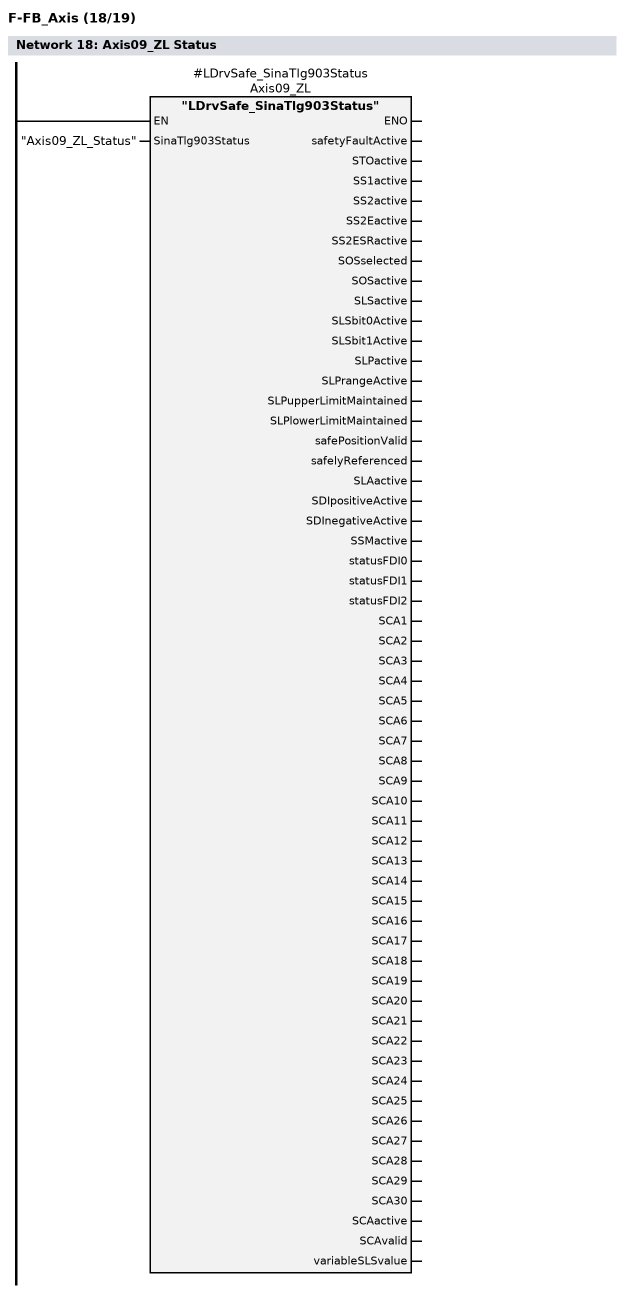
   RUNG wire#powerrail
      #LDrvSafe_SinaTlg903StatusAxis09_ZL(SinaTlg903Status := "Axis09_ZL_Status", safetyFaultActive =>, STOactive =>, SS1active =>, SS2active =>, SS2Eactive =>, SS2ESRactive =>, SOSselected =>, SOSactive =>, SLSactive =>, SLSbit0Active =>, SLSbit1Active =>, SLPactive =>, SLPrangeActive =>, SLPupperLimitMaintained =>, SLPlowerLimitMaintained =>, safePositionValid =>, safelyReferenced =>, SLAactive =>, SDIpositiveActive =>, SDInegativeActive =>, SSMactive =>, statusFDI0 =>, statusFDI1 =>, statusFDI2 =>, SCA1 =>, SCA2 =>, SCA3 =>, SCA4 =>, SCA5 =>, SCA6 =>, SCA7 =>, SCA8 =>, SCA9 =>, SCA10 =>, SCA11 =>, SCA12 =>, SCA13 =>, SCA14 =>, SCA15 =>, SCA16 =>, SCA17 =>, SCA18 =>, SCA19 =>, SCA20 =>, SCA21 =>, SCA22 =>, SCA23 =>, SCA24 =>, SCA25 =>, SCA26 =>, SCA27 =>, SCA28 =>, SCA29 =>, SCA30 =>, SCAactive =>, SCAvalid =>, variableSLSvalue =>)
   END_RUNG
   // the same network as SCL:
   #LDrvSafe_SinaTlg903StatusAxis09_ZL(SinaTlg903Status := "Axis09_ZL_Status");   // "LDrvSafe_SinaTlg903Status"
END_REGION

REGION Network 19: Axis09_ZL Control
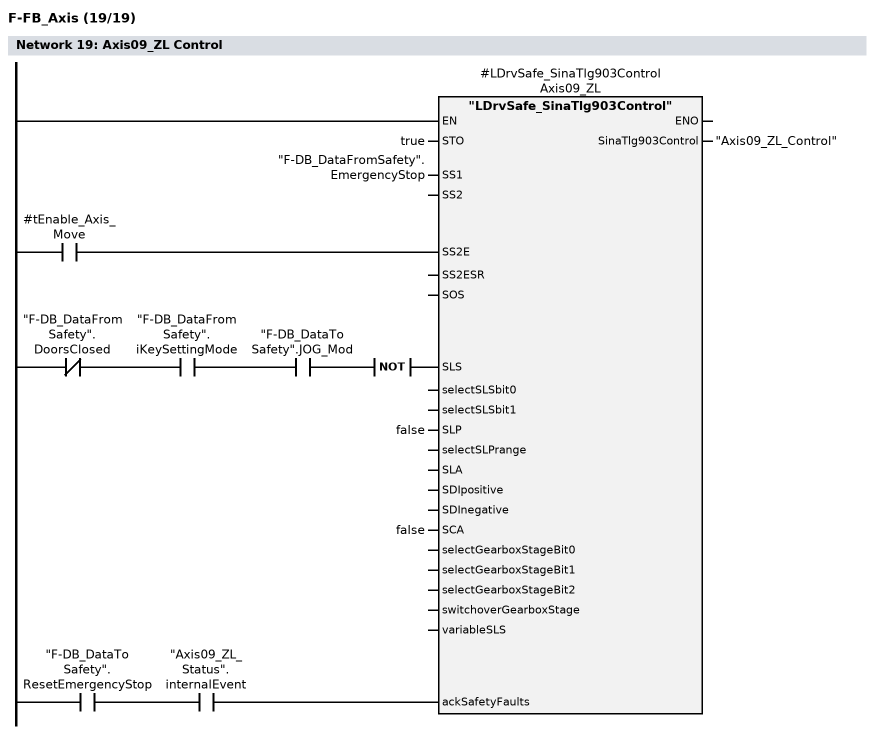
   RUNG wire#powerrail
      #LDrvSafe_SinaTlg903ControlAxis09_ZL(SS2E := wire#w1, SLS := wire#w2, ackSafetyFaults := wire#w3, STO := true, SS1 := "F-DB_DataFromSafety".EmergencyStop, SS2 :=, SS2ESR :=, SOS :=, selectSLSbit0 :=, selectSLSbit1 :=, SLP := false, selectSLPrange :=, SLA :=, SDIpositive :=, SDInegative :=, SCA := false, selectGearboxStageBit0 :=, selectGearboxStageBit1 :=, selectGearboxStageBit2 :=, switchoverGearboxStage :=, variableSLS :=, SinaTlg903Control => "Axis09_ZL_Control")
   END_RUNG
   RUNG wire#powerrail
      Contact( #tEnable_Axis_Move )
   END_RUNG wire#w1
   RUNG wire#powerrail
      I_Contact( "F-DB_DataFromSafety".DoorsClosed )
      Contact( "F-DB_DataFromSafety".iKeySettingMode )
      Contact( "F-DB_DataToSafety".JOG_Mod )
      Not()
   END_RUNG wire#w2
   RUNG wire#powerrail
      Contact( "F-DB_DataToSafety".ResetEmergencyStop )
      Contact( "Axis09_ZL_Status".internalEvent )
   END_RUNG wire#w3
   // the same network as SCL:
   #LDrvSafe_SinaTlg903ControlAxis09_ZL(STO := true,   // "LDrvSafe_SinaTlg903Control"
                           SS1 := "F-DB_DataFromSafety".EmergencyStop,
                           SS2E := #tEnable_Axis_Move,
                           SLS := NOT (NOT "F-DB_DataFromSafety".DoorsClosed AND "F-DB_DataFromSafety".iKeySettingMode AND "F-DB_DataToSafety".JOG_Mod),
                           SLP := false,
                           SCA := false,
                           ackSafetyFaults := "F-DB_DataToSafety".ResetEmergencyStop AND "Axis09_ZL_Status".internalEvent,
                           SinaTlg903Control => "Axis09_ZL_Control");
END_REGION
END_FUNCTION_BLOCK

FUNCTION_BLOCK "F-FB_Laser"   // FB140, F_LAD
{ S7_Optimized_Access := 'TRUE' }
// stored: AutoNumber false
   VAR
      FDBACK_LaserPowerSupply : FDBACK;
      FDBACK_Shutter : FDBACK;
      sFeedBackShutter : Bool;
      sAckFdbShutter : Bool;
      sLaserSupplyPower : Bool;
      sAckFdbPowLaser : Bool;
      sPositiveFrontButtonShutter : Bool;
      sNegativeFrontMaintenanceDoor : Bool;
      sNegativeFrontDoor : Bool;
      sNegativeRoofLeftDoor : Bool;
      sNegativeRoofRightDoor : Bool;
      sNegativeLaserExternDoor : Bool;
      sNegativeSasOneDoor : Bool;
   END_VAR
   VAR_TEMP   // added for the SCL form of the ladder/FBD networks
      _w1 : Bool;
      _w2 : Bool;
      _w3 : Bool;
      _w4 : Bool;
      _w5 : Bool;
      _w6 : Bool;
      _w7 : Bool;
   END_VAR
BEGIN

REGION Network 1: Laser shutter setting mode, allow opening shutter
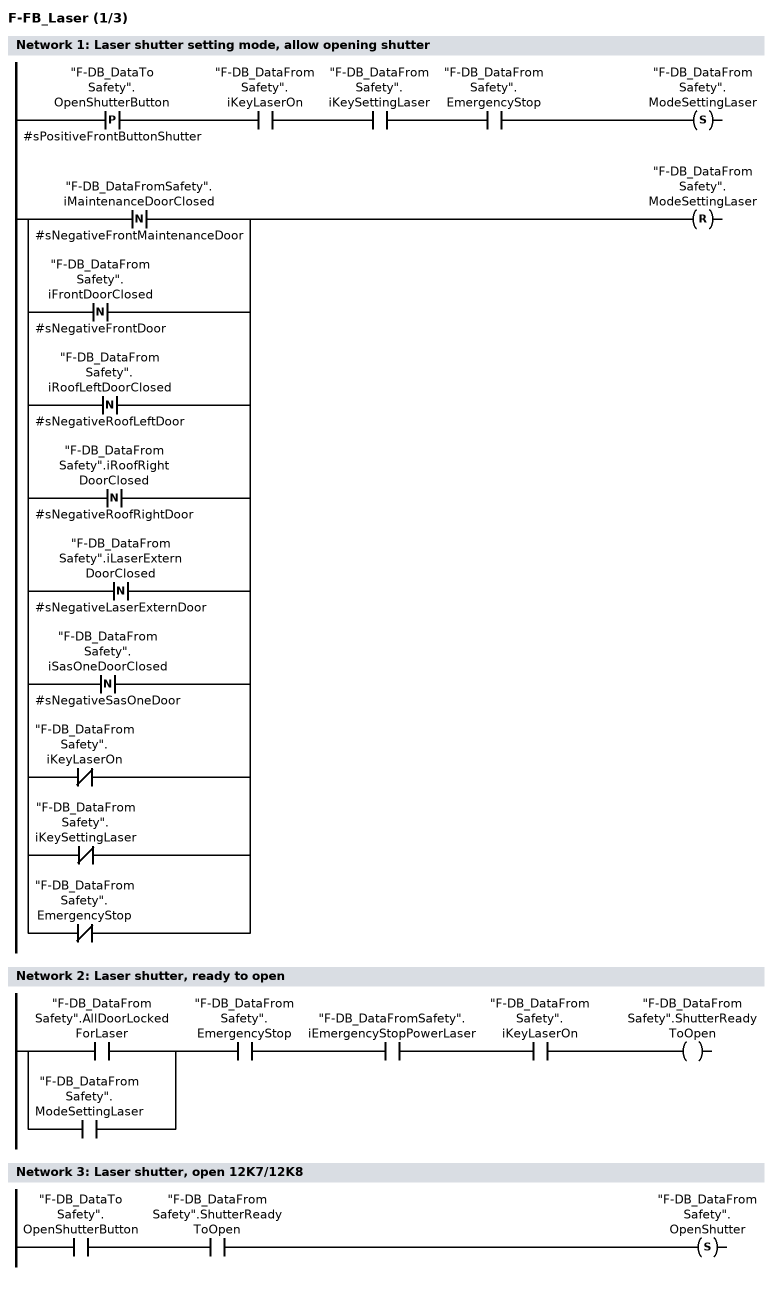
   RUNG wire#powerrail
      P_Contact(operand := "F-DB_DataToSafety".OpenShutterButton, bit := #sPositiveFrontButtonShutter)
      Contact( "F-DB_DataFromSafety".iKeyLaserOn )
      Contact( "F-DB_DataFromSafety".iKeySettingLaser )
      Contact( "F-DB_DataFromSafety".EmergencyStop )
      S_Coil( "F-DB_DataFromSafety".ModeSettingLaser )
   END_RUNG
   RUNG wire#powerrail
      N_Contact(operand := "F-DB_DataFromSafety".iMaintenanceDoorClosed, bit := #sNegativeFrontMaintenanceDoor)
      wire#w1
      R_Coil( "F-DB_DataFromSafety".ModeSettingLaser )
   END_RUNG
   RUNG wire#powerrail
      N_Contact(operand := "F-DB_DataFromSafety".iFrontDoorClosed, bit := #sNegativeFrontDoor)
   END_RUNG wire#w1
   RUNG wire#powerrail
      N_Contact(operand := "F-DB_DataFromSafety".iRoofLeftDoorClosed, bit := #sNegativeRoofLeftDoor)
   END_RUNG wire#w1
   RUNG wire#powerrail
      N_Contact(operand := "F-DB_DataFromSafety".iRoofRightDoorClosed, bit := #sNegativeRoofRightDoor)
   END_RUNG wire#w1
   RUNG wire#powerrail
      N_Contact(operand := "F-DB_DataFromSafety".iLaserExternDoorClosed, bit := #sNegativeLaserExternDoor)
   END_RUNG wire#w1
   RUNG wire#powerrail
      N_Contact(operand := "F-DB_DataFromSafety".iSasOneDoorClosed, bit := #sNegativeSasOneDoor)
   END_RUNG wire#w1
   RUNG wire#powerrail
      I_Contact( "F-DB_DataFromSafety".iKeyLaserOn )
   END_RUNG wire#w1
   RUNG wire#powerrail
      I_Contact( "F-DB_DataFromSafety".iKeySettingLaser )
   END_RUNG wire#w1
   RUNG wire#powerrail
      I_Contact( "F-DB_DataFromSafety".EmergencyStop )
   END_RUNG wire#w1
   // the same network as SCL:
   #_w1 := "F-DB_DataToSafety".OpenShutterButton AND NOT #sPositiveFrontButtonShutter;   // rising edge of "F-DB_DataToSafety".OpenShutterButton
   #sPositiveFrontButtonShutter := "F-DB_DataToSafety".OpenShutterButton;
   IF #_w1 AND "F-DB_DataFromSafety".iKeyLaserOn AND "F-DB_DataFromSafety".iKeySettingLaser AND "F-DB_DataFromSafety".EmergencyStop THEN
       "F-DB_DataFromSafety".ModeSettingLaser := TRUE;
   END_IF;
   #_w2 := NOT "F-DB_DataFromSafety".iMaintenanceDoorClosed AND #sNegativeFrontMaintenanceDoor;   // falling edge of "F-DB_DataFromSafety".iMaintenanceDoorClosed
   #sNegativeFrontMaintenanceDoor := "F-DB_DataFromSafety".iMaintenanceDoorClosed;
   #_w3 := NOT "F-DB_DataFromSafety".iFrontDoorClosed AND #sNegativeFrontDoor;   // falling edge of "F-DB_DataFromSafety".iFrontDoorClosed
   #sNegativeFrontDoor := "F-DB_DataFromSafety".iFrontDoorClosed;
   #_w4 := NOT "F-DB_DataFromSafety".iRoofLeftDoorClosed AND #sNegativeRoofLeftDoor;   // falling edge of "F-DB_DataFromSafety".iRoofLeftDoorClosed
   #sNegativeRoofLeftDoor := "F-DB_DataFromSafety".iRoofLeftDoorClosed;
   #_w5 := NOT "F-DB_DataFromSafety".iRoofRightDoorClosed AND #sNegativeRoofRightDoor;   // falling edge of "F-DB_DataFromSafety".iRoofRightDoorClosed
   #sNegativeRoofRightDoor := "F-DB_DataFromSafety".iRoofRightDoorClosed;
   #_w6 := NOT "F-DB_DataFromSafety".iLaserExternDoorClosed AND #sNegativeLaserExternDoor;   // falling edge of "F-DB_DataFromSafety".iLaserExternDoorClosed
   #sNegativeLaserExternDoor := "F-DB_DataFromSafety".iLaserExternDoorClosed;
   #_w7 := NOT "F-DB_DataFromSafety".iSasOneDoorClosed AND #sNegativeSasOneDoor;   // falling edge of "F-DB_DataFromSafety".iSasOneDoorClosed
   #sNegativeSasOneDoor := "F-DB_DataFromSafety".iSasOneDoorClosed;
   IF #_w2 OR #_w3 OR #_w4 OR #_w5 OR #_w6 OR #_w7 OR NOT "F-DB_DataFromSafety".iKeyLaserOn OR NOT "F-DB_DataFromSafety".iKeySettingLaser OR NOT "F-DB_DataFromSafety".EmergencyStop THEN
       "F-DB_DataFromSafety".ModeSettingLaser := FALSE;
   END_IF;
END_REGION

REGION Network 2: Laser shutter, ready to open
   RUNG wire#powerrail
      Contact( "F-DB_DataFromSafety".AllDoorLockedForLaser )
      wire#w1
      Contact( "F-DB_DataFromSafety".EmergencyStop )
      Contact( "F-DB_DataFromSafety".iEmergencyStopPowerLaser )
      Contact( "F-DB_DataFromSafety".iKeyLaserOn )
      Coil( "F-DB_DataFromSafety".ShutterReadyToOpen )
   END_RUNG
   RUNG wire#powerrail
      Contact( "F-DB_DataFromSafety".ModeSettingLaser )
   END_RUNG wire#w1
   // the same network as SCL:
   "F-DB_DataFromSafety".ShutterReadyToOpen := ("F-DB_DataFromSafety".AllDoorLockedForLaser OR "F-DB_DataFromSafety".ModeSettingLaser) AND "F-DB_DataFromSafety".EmergencyStop AND "F-DB_DataFromSafety".iEmergencyStopPowerLaser AND "F-DB_DataFromSafety".iKeyLaserOn;
END_REGION

REGION Network 3: Laser shutter, open 12K7/12K8
   RUNG wire#powerrail
      Contact( "F-DB_DataToSafety".OpenShutterButton )
      Contact( "F-DB_DataFromSafety".ShutterReadyToOpen )
      S_Coil( "F-DB_DataFromSafety".OpenShutter )
   END_RUNG
   // the same network as SCL:
   IF "F-DB_DataToSafety".OpenShutterButton AND "F-DB_DataFromSafety".ShutterReadyToOpen THEN
       "F-DB_DataFromSafety".OpenShutter := TRUE;
   END_IF;
END_REGION

REGION Network 4: Laser shutter, close
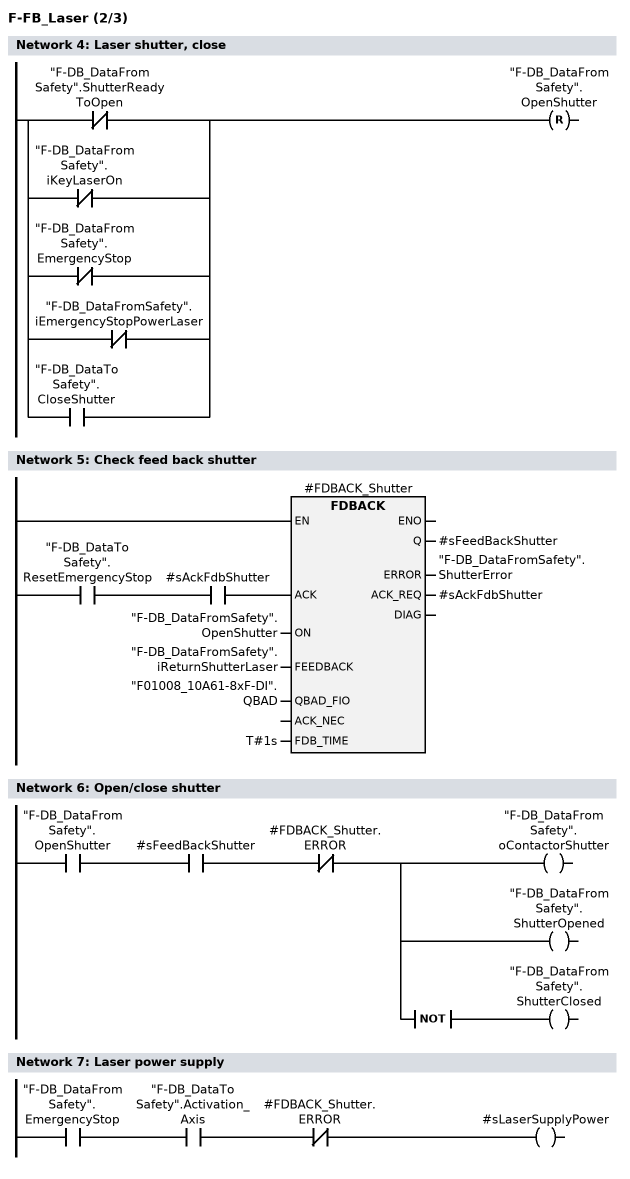
   RUNG wire#powerrail
      I_Contact( "F-DB_DataFromSafety".ShutterReadyToOpen )
      wire#w1
      R_Coil( "F-DB_DataFromSafety".OpenShutter )
   END_RUNG
   RUNG wire#powerrail
      I_Contact( "F-DB_DataFromSafety".iKeyLaserOn )
   END_RUNG wire#w1
   RUNG wire#powerrail
      I_Contact( "F-DB_DataFromSafety".EmergencyStop )
   END_RUNG wire#w1
   RUNG wire#powerrail
      I_Contact( "F-DB_DataFromSafety".iEmergencyStopPowerLaser )
   END_RUNG wire#w1
   RUNG wire#powerrail
      Contact( "F-DB_DataToSafety".CloseShutter )
   END_RUNG wire#w1
   // the same network as SCL:
   IF NOT "F-DB_DataFromSafety".ShutterReadyToOpen OR NOT "F-DB_DataFromSafety".iKeyLaserOn OR NOT "F-DB_DataFromSafety".EmergencyStop OR NOT "F-DB_DataFromSafety".iEmergencyStopPowerLaser OR "F-DB_DataToSafety".CloseShutter THEN
       "F-DB_DataFromSafety".OpenShutter := FALSE;
   END_IF;
END_REGION

REGION Network 5: Check feed back shutter
   RUNG wire#powerrail
      #FDBACK_Shutter.FDBACK(ACK := wire#w1, ON := "F-DB_DataFromSafety".OpenShutter, FEEDBACK := "F-DB_DataFromSafety".iReturnShutterLaser, QBAD_FIO := "F01008_10A61-8xF-DI".QBAD, ACK_NEC :=, FDB_TIME := T#1s, Q => #sFeedBackShutter, ERROR => "F-DB_DataFromSafety".ShutterError, ACK_REQ => #sAckFdbShutter, DIAG =>)
   END_RUNG
   RUNG wire#powerrail
      Contact( "F-DB_DataToSafety".ResetEmergencyStop )
      Contact( #sAckFdbShutter )
   END_RUNG wire#w1
   // the same network as SCL:
   #FDBACK_Shutter(ACK := "F-DB_DataToSafety".ResetEmergencyStop AND #sAckFdbShutter,   // FDBACK
                   ON := "F-DB_DataFromSafety".OpenShutter,
                   FEEDBACK := "F-DB_DataFromSafety".iReturnShutterLaser,
                   QBAD_FIO := "F01008_10A61-8xF-DI".QBAD,
                   FDB_TIME := T#1s,
                   Q => #sFeedBackShutter,
                   ERROR => "F-DB_DataFromSafety".ShutterError,
                   ACK_REQ => #sAckFdbShutter);
END_REGION

REGION Network 6: Open/close shutter
   RUNG wire#powerrail
      Contact( "F-DB_DataFromSafety".OpenShutter )
      Contact( #sFeedBackShutter )
      I_Contact( #FDBACK_Shutter.ERROR )
      wire#w1
      Coil( "F-DB_DataFromSafety".oContactorShutter )
   END_RUNG
   RUNG wire#w1
      Coil( "F-DB_DataFromSafety".ShutterOpened )
   END_RUNG
   RUNG wire#w1
      Not()
      Coil( "F-DB_DataFromSafety".ShutterClosed )
   END_RUNG
   // the same network as SCL:
   "F-DB_DataFromSafety".oContactorShutter := "F-DB_DataFromSafety".OpenShutter AND #sFeedBackShutter AND NOT #FDBACK_Shutter.ERROR;
   "F-DB_DataFromSafety".ShutterOpened := "F-DB_DataFromSafety".oContactorShutter;
   "F-DB_DataFromSafety".ShutterClosed := NOT "F-DB_DataFromSafety".oContactorShutter;
END_REGION

REGION Network 7: Laser power supply
   RUNG wire#powerrail
      Contact( "F-DB_DataFromSafety".EmergencyStop )
      Contact( "F-DB_DataToSafety".Activation_Axis )
      I_Contact( #FDBACK_Shutter.ERROR )
      Coil( #sLaserSupplyPower )
   END_RUNG
   // the same network as SCL:
   #sLaserSupplyPower := "F-DB_DataFromSafety".EmergencyStop AND "F-DB_DataToSafety".Activation_Axis AND NOT #FDBACK_Shutter.ERROR;
END_REGION

REGION Network 8: Check feed back laser power supply
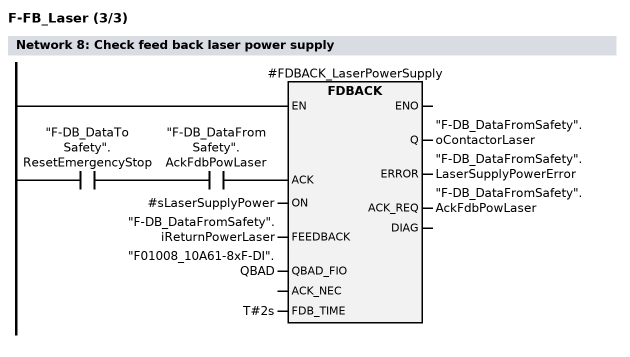
   RUNG wire#powerrail
      #FDBACK_LaserPowerSupply.FDBACK(ACK := wire#w1, ON := #sLaserSupplyPower, FEEDBACK := "F-DB_DataFromSafety".iReturnPowerLaser, QBAD_FIO := "F01008_10A61-8xF-DI".QBAD, ACK_NEC :=, FDB_TIME := T#2s, Q => "F-DB_DataFromSafety".oContactorLaser, ERROR => "F-DB_DataFromSafety".LaserSupplyPowerError, ACK_REQ => "F-DB_DataFromSafety".AckFdbPowLaser, DIAG =>)
   END_RUNG
   RUNG wire#powerrail
      Contact( "F-DB_DataToSafety".ResetEmergencyStop )
      Contact( "F-DB_DataFromSafety".AckFdbPowLaser )
   END_RUNG wire#w1
   // the same network as SCL:
   #FDBACK_LaserPowerSupply(ACK := "F-DB_DataToSafety".ResetEmergencyStop AND "F-DB_DataFromSafety".AckFdbPowLaser,   // FDBACK
                           ON := #sLaserSupplyPower,
                           FEEDBACK := "F-DB_DataFromSafety".iReturnPowerLaser,
                           QBAD_FIO := "F01008_10A61-8xF-DI".QBAD,
                           FDB_TIME := T#2s,
                           Q => "F-DB_DataFromSafety".oContactorLaser,
                           ERROR => "F-DB_DataFromSafety".LaserSupplyPowerError,
                           ACK_REQ => "F-DB_DataFromSafety".AckFdbPowLaser);
END_REGION
END_FUNCTION_BLOCK

FUNCTION_BLOCK "F-FB_DigitalOutput"   // FB111, F_LAD
{ S7_Optimized_Access := 'TRUE' }
// stored: AutoNumber false
BEGIN

REGION Network 1: Contactor for Machine
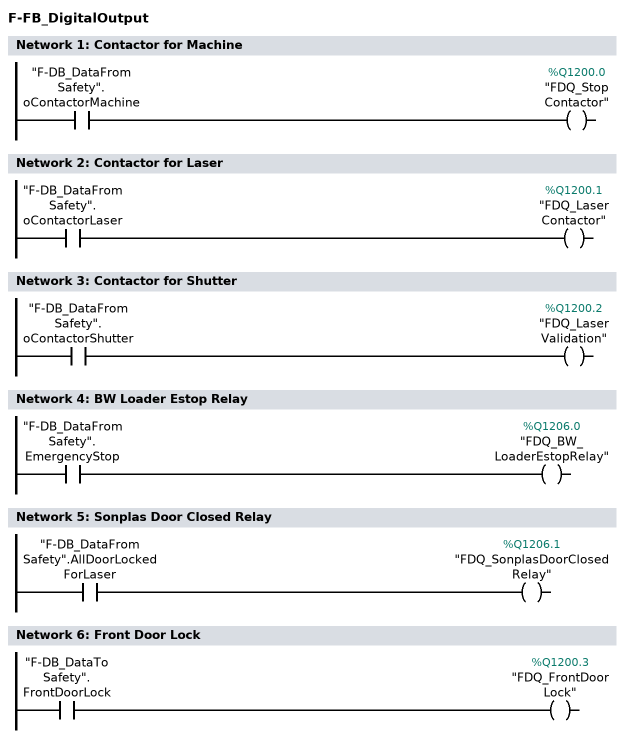
   RUNG wire#powerrail
      Contact( "F-DB_DataFromSafety".oContactorMachine )
      Coil( "FDQ_StopContactor" )
   END_RUNG
   // the same network as SCL:
   "FDQ_StopContactor" := "F-DB_DataFromSafety".oContactorMachine;
END_REGION

REGION Network 2: Contactor for Laser
   RUNG wire#powerrail
      Contact( "F-DB_DataFromSafety".oContactorLaser )
      Coil( "FDQ_LaserContactor" )
   END_RUNG
   // the same network as SCL:
   "FDQ_LaserContactor" := "F-DB_DataFromSafety".oContactorLaser;
END_REGION

REGION Network 3: Contactor for Shutter
   RUNG wire#powerrail
      Contact( "F-DB_DataFromSafety".oContactorShutter )
      Coil( "FDQ_LaserValidation" )
   END_RUNG
   // the same network as SCL:
   "FDQ_LaserValidation" := "F-DB_DataFromSafety".oContactorShutter;
END_REGION

REGION Network 4: BW Loader Estop Relay
   RUNG wire#powerrail
      Contact( "F-DB_DataFromSafety".EmergencyStop )
      Coil( "FDQ_BW_LoaderEstopRelay" )
   END_RUNG
   // the same network as SCL:
   "FDQ_BW_LoaderEstopRelay" := "F-DB_DataFromSafety".EmergencyStop;
END_REGION

REGION Network 5: Sonplas Door Closed Relay
   RUNG wire#powerrail
      Contact( "F-DB_DataFromSafety".AllDoorLockedForLaser )
      Coil( "FDQ_SonplasDoorClosedRelay" )
   END_RUNG
   // the same network as SCL:
   "FDQ_SonplasDoorClosedRelay" := "F-DB_DataFromSafety".AllDoorLockedForLaser;
END_REGION

REGION Network 6: Front Door Lock
   RUNG wire#powerrail
      Contact( "F-DB_DataToSafety".FrontDoorLock )
      Coil( "FDQ_FrontDoorLock" )
   END_RUNG
   // the same network as SCL:
   "FDQ_FrontDoorLock" := "F-DB_DataToSafety".FrontDoorLock;
END_REGION
END_FUNCTION_BLOCK

FUNCTION "FC_GestionConfigMachine" : Void   // FC33, SCL
{ S7_Optimized_Access := 'TRUE' }
// stored: SetENOAutomatically false
BEGIN
   REGION Description header 
       //==================================================================================
       // POSALUX Swiss SA / (C) Copyright 2025
       //----------------------------------------------------------------------------------
       // Title: GestionConfigMachine
       // Comment/Function: 
       //
       // Author: Fabien Waldt
       // Engineering: TIA Portal v17
       //----------------------------------------------------------------------------------
       // Change log table:
       // Version  | Date     | Expert in charge | Changes applied
       // ---------|----------|------------------|------------------------------------
       // 00.00.01 | 20250219 | WFA              | First released version
       // ==================================================================================
   END_REGION

   REGION Axis selection
       // Disable "Axis Selection" Key if not Twin Machine
       IF NOT "DB_MachineOptions".Mach_MONO_DUO THEN
           "DB_McpKeyboardSignals".sAx11_ChannelSelection.sKeyDisable := TRUE;
           "DB_McpKeyboardSignals".sAx11_ChannelSelection.sKeySWToggleStatus := FALSE;
       END_IF;
   END_REGION
END_FUNCTION

FUNCTION "FC_ResetPositionData" : Void   // FC700, SCL
{ S7_Optimized_Access := 'TRUE' }
// stored: AutoNumber false, SetENOAutomatically false
   VAR_INPUT
      iDataPosition : Int;   // Data Positions(1..5)
   END_VAR
   VAR_TEMP
      tIndex : Int;
   END_VAR
BEGIN
   REGION Description header 
       //==================================================================================
       // POSALUX Swiss SA / (C) Copyright 2025
       //----------------------------------------------------------------------------------
       // Title: FC_Fill_Data_Record
       // Comment/Function: Mise à jour des datas d'une pièce
       //
       // Author: Fabien Waldt
       // Engineering: TIA Portal v17
       //----------------------------------------------------------------------------------
       // Change log table:
       // Version  | Date     | Expert in charge | Changes applied
       // ---------|----------|------------------|------------------------------------
       // 00.00.01 | 20250224 | FWA              | First released version
       // ==================================================================================
   END_REGION
   "DB_DataPositions".Position[#iDataPosition].Part_id := 0;
       "DB_DataPositions".Position[#iDataPosition].Status := 0;
       "DB_DataPositions".Position[#iDataPosition].FailCode := 0;
       "DB_DataPositions".Position[#iDataPosition].FailCodeBackwall := 0;
       "DB_DataPositions".Position[#iDataPosition].WOZ_Status := 0;
       "DB_DataPositions".Position[#iDataPosition].WOC_Status := 0;
       "DB_DataPositions".Position[#iDataPosition].WOZ_Measure := 0.0;
       "DB_DataPositions".Position[#iDataPosition].WOC_Measure := 0;
       "DB_DataPositions".Position[#iDataPosition].TotalCycleTime := 0;
       "DB_DataPositions".Position[#iDataPosition].LaserCycleTime := 0;
       "DB_DataPositions".Position[#iDataPosition].MeasureLoadCycleTime := 0;
       FOR #tIndex := 19 TO 0 BY -1 DO
           "DB_DataPositions".Position[#iDataPosition].DMC[#tIndex] := 0;
       END_FOR;
       "DB_DataPositions".Position[#iDataPosition].OrderNbr := '---';
       "DB_DataPositions".Position[#iDataPosition].IdentNbr := '---';
       "DB_DataPositions".Position[#iDataPosition].BatchNbr := '---';
       "DB_DataPositions".Position[#iDataPosition].OperatorNbr := '---';
       "DB_DataPositions".Position[#iDataPosition].Comment := '---';
       FOR #tIndex := 0 TO 99 BY 1 DO
           "DB_DataPositions".Position[#iDataPosition].HoleSettings[#tIndex].Measure_X := 0;
           "DB_DataPositions".Position[#iDataPosition].HoleSettings[#tIndex].Measure_Y := 0;
           "DB_DataPositions".Position[#iDataPosition].HoleSettings[#tIndex].Measure_Z := 0;
           "DB_DataPositions".Position[#iDataPosition].HoleSettings[#tIndex].Measure_D := 0;
           "DB_DataPositions".Position[#iDataPosition].HoleSettings[#tIndex].Measure_Z := 0;
           "DB_DataPositions".Position[#iDataPosition].HoleSettings[#tIndex].Measure_concentricity_before := 0;
           "DB_DataPositions".Position[#iDataPosition].HoleSettings[#tIndex].Measure_concentricity_after := 0;
           "DB_DataPositions".Position[#iDataPosition].HoleSettings[#tIndex].Job_laser := 0;
       END_FOR;
END_FUNCTION

FUNCTION "FC_DataToSafety" : Void   // FC10120, SCL
{ S7_Optimized_Access := 'TRUE' }
// stored: AutoNumber false, SetENOAutomatically false
BEGIN
   REGION Transfert des datas dans le DB Buffer
       "DB_DataToSafety".OpenShutterButton := "DB_McpKeyboardSignals".sRemoteOpenShutter.sKeySWStatus;
       "DB_DataToSafety".ResetEmergencyStop := "MCP1_In".reset;
       "DB_DataToSafety".JOG_Mod := "LBP_ModeGroup".E_JOG;
       "DB_DataToSafety".Activation_Axis := "DB_DigitalOutputs".sAxisActivation.sSWStatus;
       "DB_DataToSafety".CloseShutter := "DB_DataToSafety".CloseShutter;
   END_REGION
END_FUNCTION

FUNCTION "FC_PositionCheck" : Void   // FC30, SCL
{ S7_Optimized_Access := 'TRUE' }
// stored: SetENOAutomatically false
   VAR_INPUT
      iAxisCurrentPos : LReal;
      iAxisTargetPos : LReal;
      iTolMin : Real;
      iTolMax : Real;
   END_VAR
   VAR_OUTPUT
      iInPos : Bool;
   END_VAR
BEGIN
   REGION Description header 
       //==================================================================================
       // POSALUX Swiss SA / (C) Copyright 2025
       //----------------------------------------------------------------------------------
       // Title: FC_PositionCheck
       // Comment/Function: 
       // Author: Fabien WALDT
       // Engineering: TIA Portal v17
       //----------------------------------------------------------------------------------
       // Change log table:
       // Version  | Date     | Expert in charge | Changes applied
       // ---------|----------|------------------|-----------------------------------------
       // 00.00.01 | 20250527 | WFA              | First released version
       // =================================================================================
   END_REGION

   REGION Check In Position
       IF #iAxisCurrentPos <= #iAxisTargetPos + #iTolMax
           AND #iAxisCurrentPos >= #iAxisTargetPos - #iTolMin THEN
           #iInPos := TRUE;
       ELSE
           #iInPos := FALSE;
       END_IF;
   END_REGION
END_FUNCTION

FUNCTION_BLOCK "FB_Powermeter_old"   // FB434, SCL
{ S7_Optimized_Access := 'TRUE' }
// stored: AutoNumber false, MemoryReserve 100, SetENOAutomatically false
   VAR
      sPowerMeterWorkPos : Bool;
      sPowerMeterHomePos : Bool;
      sPowerMeterToWorkMoveReq : Bool;
      sPowerMeterToHomeMoveReq : Bool;
      sPowerMeterJogMode : Bool;
      sPowermeterCylinder : "FB_CmdCylinder";
      sPowermeterInHomePos { S7_SetPoint := 'True'} : Bool;
      sPowermeterInMiddlePos : Bool;
      sPowermeterInWorkPos : Bool;
      sPowerMeterCylErrorCode : Int;
      sPowerMeterHomePosCtrlTimer : TON_TIME;
      sPowerMeterWorkPosCtrlTimer : TON_TIME;
      sMeasurePowerLaser { S7_SetPoint := 'True'} : Bool;
      sRTLaserMeasureON : R_TRIG;
      sLaserPowerValue { S7_SetPoint := 'True'} : Real;
      sWeightFactor : Real;
      sAlpha : Real;
      sDateAndTime : DTL;
      sActualMeasPower : Real;
      sTolMin : Real;
      sTolMax : Real;
      sResetMeasures : Bool;
   END_VAR
   VAR_TEMP
      tAxis01_X1SafePos : Bool;
      tLaserMeasureON : Bool;
      tActualMeasure : Int;
      tRetVal : Int;
      tAverageValue : Real;
      tStandardDeviation : Real;
      tTempReal : Real;
      tIndex : Int;
   END_VAR
   VAR CONSTANT
      POWERMETER_HOME_POS_CTRL_TIME : Time := T#6s;
      POWERMETER_WORK_POS_CTRL_TIME : Time := T#6s;
   END_VAR
BEGIN
   REGION Description header 
       //==================================================================================
       // POSALUX Swiss SA / (C) Copyright 2025
       //----------------------------------------------------------------------------------
       // Title: Initialization of axis
       // Comment/Function: 
       // Author: Fabien WALDT
       // Engineering: TIA Portal v17
       //----------------------------------------------------------------------------------
       // Change log table:
       // Version  | Date     | Expert in charge | Changes applied
       // ---------|----------|------------------|-----------------------------------------
       // 00.00.01 | 20250501 | WFA              | First released version
       // =================================================================================
   END_REGION

   REGION Axis01_X on safe position
      // Check position Axis01_X to release the powermeter
       #tAxis01_X1SafePos := "DB_AxisPosition".sAxis01_X."$AA_IM" >= "DB_AxisPosition".sAxis01_X."$MA_POS_LIMIT_PLUS" - 10.0;
   END_REGION

   REGION Blocking Axis01_X
       // Blocking Axis01_X if Powermeter is in measuring position
       "LBP_Axis01_X".A_ASpDisable := NOT #sPowerMeterHomePos OR #sPowerMeterWorkPos; 
   END_REGION

   REGION Powermeter Key / LED Management
       // Disable Powemeter Key[1] if not Jog Mode
       "DB_McpKeyboardSignals".sK1_Powermeter.sKeyDisable := NOT "LBP_ModeGroup".E_JOG OR NOT #tAxis01_X1SafePos;
       "DB_HmiKeyboardSignals".sK1_Powermeter.sKeyDisable := NOT "LBP_ModeGroup".E_JOG OR NOT #tAxis01_X1SafePos;

       // Set/Reset Toggle Powemeter Key[1]
       IF "LBP_Chan1".MDyn[92] THEN    // M92 : Powermeter to work position
           "DB_McpKeyboardSignals".sK1_Powermeter.sKeySWToggleStatus := TRUE;
           "DB_HmiKeyboardSignals".sK1_Powermeter.sKeySWToggleStatus := TRUE;
       END_IF;
       IF "LBP_Chan1".MDyn[93] OR     // M93 : Powermeter to home position
           "LBP_Chan1".A_Reset  THEN
           "DB_McpKeyboardSignals".sK1_Powermeter.sKeySWToggleStatus := FALSE;
           "DB_HmiKeyboardSignals".sK1_Powermeter.sKeySWToggleStatus := FALSE;
           END_IF;

       // Powemeter LED[1] Animation
           "DB_McpKeyboardSignals".sK1_Powermeter.sLedSWStatus :=
           ("DB_McpKeyboardSignals".sK1_Powermeter.sKeySWToggleStatus AND #tAxis01_X1SafePos)
           OR ("DB_McpKeyboardSignals".sK1_Powermeter.sKeySWToggleStatus AND "Clock_2Hz");

           "DB_HmiKeyboardSignals".sK1_Powermeter.sLedSWStatus :=
           ("DB_HmiKeyboardSignals".sK1_Powermeter.sKeySWToggleStatus AND #tAxis01_X1SafePos)
           OR ("DB_HmiKeyboardSignals".sK1_Powermeter.sKeySWToggleStatus AND "Clock_2Hz");
   END_REGION

   REGION Powermeter in work position move request
       #sPowerMeterToWorkMoveReq :=
       ("DB_McpKeyboardSignals".sK1_Powermeter.sKeySWToggleStatus AND NOT "MCP1_In".incVar)
       OR ("DB_HmiKeyboardSignals".sK1_Powermeter.sKeySWToggleStatus AND NOT "MCP1_In".incVar)
       AND ("DB_LaserMeasureZoneSwitch".sMeasure1                     // WFA Garder Sta_Meas_1 ?        // Station 1 in measure area
       AND #tAxis01_X1SafePos);
   END_REGION

   REGION Powermeter in home position move request
       #sPowerMeterToHomeMoveReq :=
       (NOT "DB_McpKeyboardSignals".sK1_Powermeter.sKeySWToggleStatus AND
        NOT "DB_HmiKeyboardSignals".sK1_Powermeter.sKeySWToggleStatus);
   END_REGION

   REGION Powermeter in JOG Mode
       #sPowerMeterJogMode := "LBP_ModeGroup".E_JOG AND "MCP1_Out".LEDincVar;
   END_REGION

   REGION Move/Control Powermeter Cylinder
       #sPowermeterCylinder(iEMinus:="DB_DigitalInputs".sPowerMeterBackCtrl.sSWStatus,
                            iEPlus:="DB_DigitalInputs".sPowerMeterFrontCtrl.sSWStatus,
                            iMinusCmd:=#sPowerMeterToHomeMoveReq,
                            iPlusCmd:=#sPowerMeterToWorkMoveReq,
                            iJOGCmd:=#sPowerMeterJogMode,
                            iMonitorTime:=T#8s,
                            ioQMinus:="DB_DigitalOutputs".sPowerMeterRetract.sSWStatus,
                            ioQPlus:="DB_DigitalOutputs".sPowerMeterAdvance.sSWStatus,
                            oMinusPos=>#sPowermeterInHomePos,
                            oMiddlePos=>#sPowermeterInMiddlePos,
                            oPlusPos=>#sPowermeterInWorkPos,
                            oErrorCode=>#sPowerMeterCylErrorCode);
   END_REGION

   REGION Powermeter Cylinder Positions
       #sPowerMeterHomePos := #sPowermeterCylinder.iEMinus;
       #sPowerMeterWorkPos := #sPowermeterCylinder.iEPlus;
   END_REGION

   REGION Powermeter Cylinder Alarms
       "LBP_AlarmMsgs".UserA[6].A70UUxx[62] := #sPowerMeterCylErrorCode = 1;    // Msg: 700662 "Alarm power meter entry"
       "LBP_AlarmMsgs".UserA[6].A70UUxx[63] := #sPowerMeterCylErrorCode = 2;    // Msg: 700663 "Alarm power meter exit"
   END_REGION

   REGION Monitoring Cylinder in home position
       #sPowerMeterHomePosCtrlTimer(IN:=#sPowerMeterToHomeMoveReq AND NOT #sPowermeterInHomePos,
                                    PT:=#POWERMETER_HOME_POS_CTRL_TIME);

       IF #sPowerMeterHomePosCtrlTimer.Q THEN
           "LBP_AlarmMsgs".ChanA[1].FDD_5C00xx[0] := TRUE;     // Msg: 510000 "Power meter runtimeerror workposition"
       END_IF;

       IF "LBP_Chan1".A_Reset THEN
           "LBP_AlarmMsgs".ChanA[1].FDD_5C00xx[0] := FALSE;    // Msg: 510000 "Power meter runtimeerror workposition"
       END_IF;

       // Read-in disable during movement
       IF #sPowerMeterToHomeMoveReq AND NOT #sPowermeterInHomePos THEN
           "LBP_AlarmMsgs".Chan[1].RID[6] := TRUE;
       END_IF;

       IF #sPowermeterInHomePos OR "LBP_Chan1".A_Reset THEN
           "LBP_AlarmMsgs".Chan[1].RID[6] := FALSE;            
       END_IF;
   END_REGION

   REGION Monitoring Cylinder in work position
       #sPowerMeterWorkPosCtrlTimer(IN := #sPowerMeterToWorkMoveReq AND NOT #sPowermeterInWorkPos,
                                    PT := #POWERMETER_WORK_POS_CTRL_TIME);

       IF #sPowerMeterWorkPosCtrlTimer.Q THEN
           "LBP_AlarmMsgs".ChanA[1].FDD_5C00xx[0] := TRUE;     // Msg: 510000 "Power meter runtimeerror workposition"
       END_IF;

       IF "LBP_Chan1".A_Reset THEN
           "LBP_AlarmMsgs".ChanA[1].FDD_5C00xx[0] := FALSE;    // Msg: 510000 "Power meter runtimeerror workposition"
       END_IF;

       // Read-in disable during movement
       IF #sPowerMeterToWorkMoveReq AND NOT #sPowermeterInWorkPos THEN
           "LBP_AlarmMsgs".Chan[1].RID[7] := TRUE;
       END_IF;

       IF #sPowermeterInWorkPos OR "LBP_Chan1".A_Reset THEN
           "LBP_AlarmMsgs".Chan[1].RID[7] := FALSE;            
       END_IF;
   END_REGION

   REGION Start/Stop measure laser power   
       // M21: Start measure laser power
       IF "LBP_Chan1".MDyn[21] THEN
           #sMeasurePowerLaser := TRUE;
       END_IF;

       // M22: Stop measure laser power
       IF "LBP_Chan1".MDyn[22] OR "MCP1_In".reset THEN
           #sMeasurePowerLaser := FALSE;
       END_IF;
   END_REGION

   REGION Power value calculation  
       #tLaserMeasureON := #sMeasurePowerLaser OR #sPowerMeterJogMode;

       // Init Powermeter value when restart
       #sRTLaserMeasureON(CLK:=#tLaserMeasureON AND #sPowermeterInWorkPos);
       IF #sRTLaserMeasureON.Q THEN
           #sLaserPowerValue := 0.0;
       END_IF;

       // Power value calculation
       IF #tLaserMeasureON AND #sPowermeterInWorkPos THEN
           #sLaserPowerValue := #sAlpha * "DB_AnalogInputs".sLaserPowerMeter.sSWRealValue +
           (1 - #sAlpha) * #sLaserPowerValue;
           "LBP_NC".A_Setval_anaIn3 := DINT_TO_WORD(REAL_TO_DINT(#sLaserPowerValue * #sWeightFactor));
           "LBP_NC".A_InMask_anaIn3 := TRUE;
       END_IF;
   END_REGION

   REGION Date et Time reading
       #tRetVal := RD_SYS_T(OUT => #sDateAndTime);
   END_REGION

   REGION Measurement archiving
       IF "LBP_Chan1".MDyn[39] THEN
           #tActualMeasure := "DB_PowermeterMeasures".ActualMeasure + 1;
           IF #tActualMeasure >= "DB_PowermeterMeasures".NbMeasure THEN
               #tActualMeasure := 0;
               "DB_PowermeterMeasures".Table_full := TRUE;  // WFA Bit jamais remis à 0
           END_IF;

           "DB_PowermeterMeasures".Measures[#tActualMeasure].Day_meas := DTL_TO_DATE(#sDateAndTime);
           "DB_PowermeterMeasures".Measures[#tActualMeasure].Time_day := DTL_TO_TOD(#sDateAndTime);

           #sActualMeasPower := "LBP_Chan1".H1;

           "DB_PowermeterMeasures".ActualTotalMeas :=
           #sActualMeasPower
           - "DB_PowermeterMeasures".Measures[#tActualMeasure].ValuePower
           + "DB_PowermeterMeasures".ActualTotalMeas;

           "DB_PowermeterMeasures".Measures[#tActualMeasure].ValuePower := #sActualMeasPower;

           REGION Average and Standard Deviation Calculation
               IF "DB_PowermeterMeasures".Table_full THEN
                   #tActualMeasure := 100;
               ELSIF #tActualMeasure < 0 THEN
                   #tActualMeasure := 1;
               END_IF;

               #tAverageValue := "DB_PowermeterMeasures".ActualTotalMeas / #tActualMeasure;

               #tTempReal := ((#tAverageValue * -2.0 * "DB_PowermeterMeasures".ActualTotalMeas) / #tActualMeasure) + #tAverageValue;

               #tStandardDeviation := SQRT(("DB_PowermeterMeasures".ActualMeasure * "DB_PowermeterMeasures".ActualMeasure / #tActualMeasure) + #tTempReal);
           END_REGION

           REGION Compute CM  (" Tol+" - " Tol-" ) / (6 Sigma) process capability index
               IF #tStandardDeviation * 6.0 > 0.0001 THEN
                   #tTempReal := #tStandardDeviation;
               ELSE
                   #tTempReal := 1.0;
               END_IF;

               "DB_PowermeterMeasures".Measures[#tActualMeasure].ValueCM :=
               (#sTolMax - #sTolMin) / #tTempReal;

               "DB_PowermeterMeasures".ActualMeasure := #tActualMeasure;
           END_REGION
       END_IF;
   END_REGION

   REGION Reset Measures
       IF #sResetMeasures THEN
           FOR #tIndex := 0 TO "DB_PowermeterMeasures".NbMeasure - 1 DO
               "DB_PowermeterMeasures".Measures[#tIndex].Job_meas := -1;
               "DB_PowermeterMeasures".Measures[#tIndex].ValuePower := 0.0;
               "DB_PowermeterMeasures".Measures[#tIndex].ValueCM := 0.0;
           END_FOR;
       END_IF;
   END_REGION
END_FUNCTION_BLOCK

FUNCTION "LBP_CallBackAuxFunc" : Void   // FC12, SCL
TITLE = Auxiliary functions / Fonctions auxiliaires
{ S7_Optimized_Access := 'FALSE' }
AUTHOR : SINUMERIK
FAMILY : SINUMERIK_ONE
VERSION : 6.24
// Call interface for users for auxiliary functions, the block is called on an event-driven basis in the basic program when new auxiliary functions are available / Interface d'appel pour utilisateurs de fonctions auxiliaires. Le bloc est appelé dans le programme de base sur événement lorsque de nouvelles fonctions auxiliaires sont disponibles
// stored: AutoNumber false, IsIECCheckEnabled true, SetENOAutomatically false
   VAR_INPUT
      Chan : Byte;   // Index of channel / Indice de canal
   END_VAR
BEGIN
END_FUNCTION

FUNCTION "FC_AnalogInputsInit" : Void   // FC31, SCL
{ S7_Optimized_Access := 'TRUE' }
// stored: AutoNumber false, SetENOAutomatically false
   VAR_TEMP
      tBusy : Bool;
      tRetVal : Int;
   END_VAR
BEGIN
   REGION Description header 
       //==================================================================================
       // POSALUX Swiss SA / (C) Copyright 2025
       //----------------------------------------------------------------------------------
       // Title: Analog Inputs Initialisation 
       // Comment/Function: Initialisation of analog inputs
       // Author: Fabien WALDT
       // Engineering: TIA Portal v17
       //----------------------------------------------------------------------------------
       // Change log table:
       // Version  | Date     | Expert in charge | Changes applied
       // ---------|----------|------------------|-----------------------------------------
       // 00.00.01 | 20250423 | WFA              | First released version
       // =================================================================================
   END_REGION
   // Transfert Data From PLC to IHM at Start
   IF "FirstScan" THEN
       "DB_AnalogInputs".sLaserPowerMeter.sDownload := TRUE;
       "DB_AnalogInputs".sAxisB_ClampingPart.sDownload := TRUE;
       "DB_AnalogInputs".sLaserAirPressureProcess.sDownload := TRUE;
       "DB_AnalogInputs".sInletAirPressure.sDownload := TRUE;
       "DB_AnalogInputs".sAmbiantTemperature.sDownload := TRUE;
       "DB_AnalogInputs".sMachineTemperature.sDownload := TRUE;
       "DB_AnalogInputs".sCold_WaterTemperatureInput.sDownload := TRUE;
       "DB_AnalogInputs".sCold_WaterTemperatureOutput.sDownload := TRUE;
       "DB_AnalogInputs".sX_AxisTemperaturePT1000.sDownload := TRUE;
       "DB_AnalogInputs".sY_AxisTemperaturePT1000.sDownload := TRUE;
       "DB_AnalogInputs".sX_AxisTemperaturePTC.sDownload := TRUE;
       "DB_AnalogInputs".sY_AxisTemperaturePTC.sDownload := TRUE;
       "DB_AnalogInputs".sNozzleOverpressure.sDownload := TRUE;
       "DB_AnalogInputs".sOpticalPathOverpressure.sDownload := TRUE;
       "DB_AnalogInputs".sLaserHeadOverpressure.sDownload := TRUE;
       "DB_AnalogInputs".sZLAxisOverpressure.sDownload := TRUE;
       "DB_AnalogInputs".sXYAxisOverpressure.sDownload := TRUE;
       "DB_AnalogInputs".sLeftAspiration.sDownload := TRUE;
       "DB_AnalogInputs".sRightAspiration.sDownload := TRUE;
       "DB_AnalogInputs".sClimTemperature.sDownload := TRUE;
       "DB_AnalogInputs".sSensorControllerStation1.sDownload := TRUE;
       "DB_AnalogInputs".sCabinetTemperature.sDownload := TRUE;
   END_IF;

   // Update data from IHM
   IF "DB_OPC_AnalogInputs".Update THEN
       "DB_OPC_AnalogInputs".Signals["DB_OPC_AnalogInputs".Parameters.ItemNumber].Delay := LREAL_TO_REAL("DB_OPC_AnalogInputs".Parameters.Delay);
       "DB_OPC_AnalogInputs".Signals["DB_OPC_AnalogInputs".Parameters.ItemNumber].DiffErrorMax := LREAL_TO_REAL("DB_OPC_AnalogInputs".Parameters.DiffErrorMax);
       "DB_OPC_AnalogInputs".Signals["DB_OPC_AnalogInputs".Parameters.ItemNumber].DiffErrorMin := LREAL_TO_REAL("DB_OPC_AnalogInputs".Parameters.DiffErrorMin);
       "DB_OPC_AnalogInputs".Signals["DB_OPC_AnalogInputs".Parameters.ItemNumber].DiffWarnMax := LREAL_TO_REAL("DB_OPC_AnalogInputs".Parameters.DiffWarnMax);
       "DB_OPC_AnalogInputs".Signals["DB_OPC_AnalogInputs".Parameters.ItemNumber].DiffWarnMin := LREAL_TO_REAL("DB_OPC_AnalogInputs".Parameters.DiffWarnMin);
       "DB_OPC_AnalogInputs".Signals["DB_OPC_AnalogInputs".Parameters.ItemNumber].Id := DINT_TO_INT("DB_OPC_AnalogInputs".Parameters.Id);
       "DB_OPC_AnalogInputs".Signals["DB_OPC_AnalogInputs".Parameters.ItemNumber].Offset := LREAL_TO_REAL("DB_OPC_AnalogInputs".Parameters.Offset);
       "DB_OPC_AnalogInputs".Signals["DB_OPC_AnalogInputs".Parameters.ItemNumber].Gain := LREAL_TO_REAL("DB_OPC_AnalogInputs".Parameters.Gain);
       "DB_OPC_AnalogInputs".Signals["DB_OPC_AnalogInputs".Parameters.ItemNumber].Target := LREAL_TO_REAL("DB_OPC_AnalogInputs".Parameters.Target);

       "DB_OPC_AnalogInputs".Signals["DB_OPC_AnalogInputs".Parameters.ItemNumber].Update := TRUE;
       "DB_OPC_AnalogInputs".Update := FALSE;
   END_IF;

   // Permet de copier les valeurs en cours dans les valeurs initiales (A utiliser avec précautions)
   #tRetVal := WRIT_DBL(REQ := FALSE,
            SRCBLK := "DB_AnalogInputDataHMI",
            BUSY => #tBusy,
            DSTBLK => "DB_AnalogInputDataHMI");
END_FUNCTION

FUNCTION_BLOCK "FB_ChillerSMC"   // FB541, SCL
{ S7_Optimized_Access := 'TRUE' }
// stored: AutoNumber false, MemoryReserve 100, SetENOAutomatically false
   VAR
      sTimeHeadChillerCutOff { S7_SetPoint := 'True'} : TON_TIME;
      sTimeHeadChillerTemperature { S7_SetPoint := 'True'} : TON_TIME;
      sTimeSourceChillerCutOff { S7_SetPoint := 'True'} : TON_TIME;
      sTimeSourceChillerTemperature { S7_SetPoint := 'True'} : TON_TIME;
   END_VAR
   VAR CONSTANT
      TIME_CHILLER_CUTOFF : Time := T#8s;
      TIME_CHILLER_TEMPERATURE : Time := T#8s;
   END_VAR
BEGIN
   REGION Description header 
       //==================================================================================
       // POSALUX Swiss SA / (C) Copyright 2025
       //----------------------------------------------------------------------------------
       // Title: FB_Chiller_SMC
       // Comment/Function:
       // Author: Fabien Waldt
       // Engineering: TIA Portal v19
       //----------------------------------------------------------------------------------
       // Change log table:
       // Version  | Date     | Expert in charge | Changes applied
       // ---------|----------|------------------|------------------------------------
       // 00.00.01 | 20250904 | FWA              | First released version
       // ==================================================================================
   END_REGION

   REGION Head Chiller
       REGION Alarm Head Chiller : CutOff
           #sTimeHeadChillerCutOff(IN := "DB_PowerOn".sMachineReadySoft AND NOT "DB_DigitalInputs".sHeadChillerCutOff.sSWStatus,
                                   PT := #TIME_CHILLER_CUTOFF,
                                   Q => "LBP_AlarmMsgs".UserA[02].A70UUxx[28]);
       END_REGION

       REGION Alarm Head Chiller : Temperature
           #sTimeHeadChillerTemperature(IN := "DB_PowerOn".sMachineReadySoft AND NOT "DB_DigitalInputs".sHeadChillerTemperature.sSWStatus,
                                        PT := #TIME_CHILLER_TEMPERATURE,
                                        Q => "LBP_AlarmMsgs".UserA[02].A70UUxx[29]);
       END_REGION
   END_REGION

   REGION Source Chiller
       REGION Alarm Source Chiller : CutOff
           #sTimeSourceChillerCutOff(IN := "DB_PowerOn".sMachineReadySoft AND NOT "DB_DigitalInputs".sSourceChillerCutOff.sSWStatus,
                                     PT := #TIME_CHILLER_CUTOFF,
                                     Q => "LBP_AlarmMsgs".UserA[02].A70UUxx[30]);
       END_REGION

       REGION Alarm Source Chiller : Temperature
           #sTimeSourceChillerTemperature(IN := "DB_PowerOn".sMachineReadySoft AND NOT "DB_DigitalInputs".sSourceChillerTemperature.sSWStatus,
                                          PT := #TIME_CHILLER_TEMPERATURE,
                                          Q => "LBP_AlarmMsgs".UserA[02].A70UUxx[31]);
       END_REGION
   END_REGION
END_FUNCTION_BLOCK

FUNCTION_BLOCK "FB_ChillerTermotek"   // FB540, SCL
{ S7_Optimized_Access := 'TRUE' }
// stored: AutoNumber false, MemoryReserve 100, SetENOAutomatically false
   VAR
      sTimeHeadChillerHighPressure { S7_SetPoint := 'True'} : TON_TIME;
      sTimeHeadChillerWaterTemperature { S7_SetPoint := 'True'} : TON_TIME;
      sTimeHeadChillerAmbiantTemperature { S7_SetPoint := 'True'} : TON_TIME;
      sTimeOutFlowHeadChiller : TON_TIME;
      sTimeOutLevelHeadChiller { S7_SetPoint := 'True'} : TON_TIME;
      sTimeOutHeadChillerGood : TON_TIME;
      sTimeSourceChillerHighPressure { S7_SetPoint := 'True'} : TON_TIME;
      sTimeSourceChillerWaterTemperature { S7_SetPoint := 'True'} : TON_TIME;
      sTimeSourceChillerAmbiantTemperature { S7_SetPoint := 'True'} : TON_TIME;
      sTimeOutFlowSourceChiller : TON_TIME;
      sTimeOutLevelSourceChiller { S7_SetPoint := 'True'} : TON_TIME;
      sTimeOutSourceChillerGood : TON_TIME;
   END_VAR
   VAR CONSTANT
      TIME_CHILLER_HIGH_PRESSURE : Time := T#8s;
      TIME_CHILLER_WATER_TEMPERATURE : Time := T#8s;
      TIME_CHILLER_AMBIANT_TEMPERATURE : Time := T#8s;
      TIME_OUT_FLOW_CHILLER : Time := T#8S;
      TIME_OUT_LEVEL_CHILLER : Time := T#8S;
      TIME_OUT_CHILLER_GOOD : Time := T#8S;
   END_VAR
BEGIN
   REGION Description header 
       //==================================================================================
       // POSALUX Swiss SA / (C) Copyright 2025
       //----------------------------------------------------------------------------------
       // Title: FB_Chiller_Termotek
       // Comment/Function:
       // Author: Fabien Waldt
       // Engineering: TIA Portal v19
       //----------------------------------------------------------------------------------
       // Change log table:
       // Version  | Date     | Expert in charge | Changes applied
       // ---------|----------|------------------|------------------------------------
       // 00.00.01 | 20250904 | FWA              | First released version
       // ==================================================================================
   END_REGION

   REGION Head Chiller
       REGION Alarm Head Chiller : High Pressure
           #sTimeHeadChillerHighPressure(IN := "DB_PowerOn".sMachineReadySoft AND NOT "DB_DigitalInputs".sHeadChillerHighPressure.sSWStatus,
                                     PT := #TIME_CHILLER_HIGH_PRESSURE,
                                     Q => "LBP_AlarmMsgs".UserA[02].A70UUxx[04]);
       END_REGION

       REGION Alarm Head Chiller : Water Temperature
           #sTimeHeadChillerWaterTemperature(IN := "DB_PowerOn".sMachineReadySoft AND NOT "DB_DigitalInputs".sHeadChillerWaterTemperature.sSWStatus,
                                         PT := #TIME_CHILLER_WATER_TEMPERATURE,
                                         Q => "LBP_AlarmMsgs".UserA[02].A70UUxx[05]);
       END_REGION

       REGION Alarm Head Chiller : Ambiant Temperature
           #sTimeHeadChillerAmbiantTemperature(IN := "DB_PowerOn".sMachineReadySoft AND NOT "DB_DigitalInputs".sHeadChillerAmbiantTemperature.sSWStatus,
                                           PT := #TIME_CHILLER_AMBIANT_TEMPERATURE,
                                           Q => "LBP_AlarmMsgs".UserA[02].A70UUxx[06]);
       END_REGION

       REGION Alarm Head chiller : water flow error
           #sTimeOutFlowHeadChiller(IN := "DB_PowerOn".sMachineReadySoft AND NOT "DB_DigitalInputs".sHeadChillerFlow.sSWStatus,
                                PT := #TIME_OUT_FLOW_CHILLER,
                                Q => "LBP_AlarmMsgs".UserA[2].A70UUxx[0]);
       END_REGION

       REGION Alarm Head chiller : faulty
           #sTimeOutLevelHeadChiller(IN := "DB_PowerOn".sMachineReadySoft AND NOT "DB_DigitalInputs".sHeadChillerCollectivFault.sSWStatus,
                                 PT := #TIME_OUT_LEVEL_CHILLER,
                                 Q => "LBP_AlarmMsgs".UserA[2].A70UUxx[1]);
       END_REGION

       REGION Alarm Head chiller : water level error
           #sTimeOutHeadChillerGood(IN := "DB_PowerOn".sMachineReadySoft AND NOT "DB_DigitalInputs".sHeadChillerWaterLevel.sSWStatus,
                                PT := #TIME_OUT_CHILLER_GOOD,
                                Q => "LBP_AlarmMsgs".UserA[2].A70UUxx[2]);
       END_REGION
   END_REGION

   REGION Source Chiller
       REGION Alarm Source Chiller : High Pressure
           #sTimeSourceChillerHighPressure(IN := "DB_PowerOn".sMachineReadySoft AND NOT "DB_DigitalInputs".sSourceChillerHighPressure.sSWStatus,
                                           PT := #TIME_CHILLER_HIGH_PRESSURE,
                                           Q => "LBP_AlarmMsgs".UserA[02].A70UUxx[10]);
       END_REGION

       REGION Alarm Source Chiller : Water Temperature
          #sTimeSourceChillerWaterTemperature(IN := "DB_PowerOn".sMachineReadySoft AND NOT "DB_DigitalInputs".sSourceChillerWaterTemperature.sSWStatus,
                                              PT := #TIME_CHILLER_WATER_TEMPERATURE,
                                              Q => "LBP_AlarmMsgs".UserA[02].A70UUxx[11]);
       END_REGION

       REGION Alarm Source Chiller : Ambiant Temperature
           #sTimeSourceChillerAmbiantTemperature(IN := "DB_PowerOn".sMachineReadySoft AND NOT "DB_DigitalInputs".sSourceChillerAmbiantTemperature.sSWStatus,
                                                 PT := #TIME_CHILLER_AMBIANT_TEMPERATURE,
                                                 Q => "LBP_AlarmMsgs".UserA[02].A70UUxx[12]);
       END_REGION

       REGION Alarm Source chiller : water flow error
           #sTimeOutFlowSourceChiller(IN := "DB_PowerOn".sMachineReadySoft AND NOT "DB_DigitalInputs".sSourceChillerFlow.sSWStatus,
                                      PT := #TIME_OUT_FLOW_CHILLER,
                                      Q => "LBP_AlarmMsgs".UserA[2].A70UUxx[7]);
       END_REGION

       REGION Alarm Source chiller : faulty
           #sTimeOutLevelSourceChiller(IN := "DB_PowerOn".sMachineReadySoft AND NOT "DB_DigitalInputs".sSourceChillerWaterLevel.sSWStatus,
                                       PT := #TIME_OUT_LEVEL_CHILLER,
                                       Q => "LBP_AlarmMsgs".UserA[2].A70UUxx[8]);
       END_REGION

       REGION Alarm Source chiller : water level error
           #sTimeOutSourceChillerGood(IN := "DB_PowerOn".sMachineReadySoft AND NOT "DB_DigitalInputs".sSourceChillerCollectivFault.sSWStatus,
                                      PT := #TIME_OUT_CHILLER_GOOD,
                                      Q => "LBP_AlarmMsgs".UserA[2].A70UUxx[9]);
       END_REGION
   END_REGION
END_FUNCTION_BLOCK

FUNCTION "FC_ChillerMain" : Void   // FC540, SCL
{ S7_Optimized_Access := 'TRUE' }
// stored: AutoNumber false, SetENOAutomatically false
BEGIN
   REGION Description header 
       //==================================================================================
       // POSALUX Swiss SA / (C) Copyright 2025
       //----------------------------------------------------------------------------------
       // Title: FC_Chiller_Main
       // Comment/Function:
       // Author: Fabien Waldt
       // Engineering: TIA Portal v19
       //----------------------------------------------------------------------------------
       // Change log table:
       // Version  | Date     | Expert in charge | Changes applied
       // ---------|----------|------------------|------------------------------------
       // 00.00.01 | 20250904 | FWA              | First released version
       // ==================================================================================
   END_REGION

   REGION Option Chiller : TERMOTEK
       IF "DB_MachineOptions".Chiller.Termotek THEN
           "DB_ChillerTermotek"();
       END_IF;
   END_REGION

   REGION Option Chiller : SMC
       IF "DB_MachineOptions".Chiller.SMC THEN
           "DB_ChillerSMC"();
       END_IF;
   END_REGION
END_FUNCTION

FUNCTION "FC_AnalogInputAction" : Void   // FC1302, SCL
{ S7_Optimized_Access := 'TRUE' }
// stored: AutoNumber false, SetENOAutomatically false
   VAR_INPUT
      iReset : Bool;
   END_VAR
   VAR_OUTPUT
      oBadPartOnFixture : Bool;
      oID_MeasureBad : Int;
   END_VAR
   VAR_TEMP
      tIndex : Int;
      tResultByte0 : Int;
      tResultByte2 : Int;
      tResultByte3 : Int;
      tInitValue : LWord;
   END_VAR
BEGIN
   REGION Description header 
       //==================================================================================
       // POSALUX Swiss SA / (C) Copyright 2025
       //----------------------------------------------------------------------------------
       // Title: FC_PLC-ISO-IHM
       // Comment/Function: Manage analog variables
       //                   - BadPartOnFixture:  Set to 1 if any BadPartOnFixture bit in DB_Analog_Input_Setting = 1  
       //                                        Set to 0 if all BadPartOnFixture bits in DB_Analog_Input_Setting = 0  
       // Author: Fabien Waldt
       // Engineering: TIA Portal v17
       //----------------------------------------------------------------------------------
       // Change log table:
       // Version  | Date     | Expert in charge | Changes applied
       // ---------|----------|------------------|------------------------------------
       // 00.00.01 | 20250312 | WFA              | First released version
       // 00.00.02 | 20250807 | WFA              | Removal of the StopMachine feature
       // ==================================================================================
   END_REGION

   REGION Reset Values
       IF #iReset THEN
           #tInitValue := 0;
           FOR #tIndex := 0 TO 74 DO
               POKE(area := 16#84,
                    dbNumber := 1304,
                    byteOffset := #tIndex,
                    value := #tInitValue);
           END_FOR;
       END_IF;
   END_REGION

   REGION Bad Part On Fixture
       FOR #tIndex := 0 TO 74 BY 4 DO
           #tResultByte0 := PEEK(area := 16#84, dbNumber := 1304, byteOffset := #tIndex);
           #tResultByte2 := PEEK(area := 16#84, dbNumber := 1304, byteOffset := #tIndex + 2);
           #tResultByte3 := PEEK(area := 16#84, dbNumber := 1304, byteOffset := #tIndex + 3);
           #oBadPartOnFixture := FALSE;
           IF #tResultByte0.%X0 THEN
               #oBadPartOnFixture := TRUE;
               #oID_MeasureBad := ABS(SHL(IN := #tResultByte2, N := 8) OR #tResultByte3);
               EXIT;
           END_IF;
       END_FOR;
   END_REGION
END_FUNCTION

FUNCTION "FC_AnalogInputConfig" : Void   // FC35, SCL
{ S7_Optimized_Access := 'TRUE' }
// stored: SetENOAutomatically false
BEGIN
   REGION Description header 
       //==================================================================================
       // POSALUX Swiss SA / (C) Copyright 2025
       //----------------------------------------------------------------------------------
       // Title: FC_AnalogInputConfig
       // Comment/Function:
       //
       // Author: Fabien Waldt
       // Engineering: TIA Portal v17
       //----------------------------------------------------------------------------------
       // Change log table:
       // Version  | Date     | Expert in charge | Changes applied
       // ---------|----------|------------------|------------------------------------
       // 00.00.01 | 20250312 | WFA              | First released version
       // ==================================================================================
   END_REGION

   REGION Laser_Power_Meter
       "DB_AnalogInputDataPLC".Laser_Power_Meter.EnableAlarmMin   := FALSE;
       "DB_AnalogInputDataPLC".Laser_Power_Meter.EnableWarningMin := FALSE;
       "DB_AnalogInputDataPLC".Laser_Power_Meter.EnableWarningMax := FALSE;
       "DB_AnalogInputDataPLC".Laser_Power_Meter.EnableAlarmMax   := FALSE;
   END_REGION

   REGION Axis_B_Clamping_Part
       "DB_AnalogInputDataPLC".Axis_B_Clamping_Part.EnableAlarmMin   := FALSE;
       "DB_AnalogInputDataPLC".Axis_B_Clamping_Part.EnableWarningMin := FALSE;
       "DB_AnalogInputDataPLC".Axis_B_Clamping_Part.EnableWarningMax := FALSE;
       "DB_AnalogInputDataPLC".Axis_B_Clamping_Part.EnableAlarmMax   := FALSE;
   END_REGION

   REGION Laser_Air_Pressure_Process
       "DB_AnalogInputDataPLC".Laser_Air_Pressure_Process.EnableAlarmMin   := TRUE;
       "DB_AnalogInputDataPLC".Laser_Air_Pressure_Process.EnableWarningMin := TRUE;
       "DB_AnalogInputDataPLC".Laser_Air_Pressure_Process.EnableWarningMax := TRUE;
       "DB_AnalogInputDataPLC".Laser_Air_Pressure_Process.EnableAlarmMax   := TRUE;
   END_REGION

   REGION Inlet_Air_Pressure
       "DB_AnalogInputDataPLC".Inlet_Air_Pressure.EnableAlarmMin   := TRUE;
       "DB_AnalogInputDataPLC".Inlet_Air_Pressure.EnableWarningMin := TRUE;
       "DB_AnalogInputDataPLC".Inlet_Air_Pressure.EnableWarningMax := TRUE;
       "DB_AnalogInputDataPLC".Inlet_Air_Pressure.EnableAlarmMax   := TRUE;
   END_REGION

   REGION Ambiant_Temperature
       "DB_AnalogInputDataPLC".Ambiant_Temperature.EnableAlarmMin   := TRUE;
       "DB_AnalogInputDataPLC".Ambiant_Temperature.EnableWarningMin := TRUE;
       "DB_AnalogInputDataPLC".Ambiant_Temperature.EnableWarningMax := TRUE;
       "DB_AnalogInputDataPLC".Ambiant_Temperature.EnableAlarmMax   := TRUE;
   END_REGION

   REGION Machine_Temperature
       "DB_AnalogInputDataPLC".Machine_Temperature.EnableAlarmMin   := TRUE;
       "DB_AnalogInputDataPLC".Machine_Temperature.EnableWarningMin := TRUE;
       "DB_AnalogInputDataPLC".Machine_Temperature.EnableWarningMax := TRUE;
       "DB_AnalogInputDataPLC".Machine_Temperature.EnableAlarmMax   := TRUE;
   END_REGION

   REGION Cold_Water_Temperature_Input
       "DB_AnalogInputDataPLC".Cold_Water_Temperature_Input.EnableAlarmMin   := TRUE;
       "DB_AnalogInputDataPLC".Cold_Water_Temperature_Input.EnableWarningMin := TRUE;
       "DB_AnalogInputDataPLC".Cold_Water_Temperature_Input.EnableWarningMax := TRUE;
       "DB_AnalogInputDataPLC".Cold_Water_Temperature_Input.EnableAlarmMax   := TRUE;
   END_REGION

   REGION Cold_Water_Temperature_Output
       "DB_AnalogInputDataPLC".Cold_Water_Temperature_Output.EnableAlarmMin   := TRUE;
       "DB_AnalogInputDataPLC".Cold_Water_Temperature_Output.EnableWarningMin := TRUE;
       "DB_AnalogInputDataPLC".Cold_Water_Temperature_Output.EnableWarningMax := TRUE;
       "DB_AnalogInputDataPLC".Cold_Water_Temperature_Output.EnableAlarmMax   := TRUE;
   END_REGION

   REGION X_Axis_Temperature_PT1000
       "DB_AnalogInputDataPLC".X_Axis_Temperature_PT1000.EnableAlarmMin   := FALSE; //WFA
       "DB_AnalogInputDataPLC".X_Axis_Temperature_PT1000.EnableWarningMin := FALSE; //WFA
       "DB_AnalogInputDataPLC".X_Axis_Temperature_PT1000.EnableWarningMax := TRUE;
       "DB_AnalogInputDataPLC".X_Axis_Temperature_PT1000.EnableAlarmMax   := TRUE;
   END_REGION

   REGION Y_Axis_Temperature_PT1000
       "DB_AnalogInputDataPLC".Y_Axis_Temperature_PT1000.EnableAlarmMin   := FALSE; //WFA
       "DB_AnalogInputDataPLC".Y_Axis_Temperature_PT1000.EnableWarningMin := FALSE; //WFA
       "DB_AnalogInputDataPLC".Y_Axis_Temperature_PT1000.EnableWarningMax := TRUE;
       "DB_AnalogInputDataPLC".Y_Axis_Temperature_PT1000.EnableAlarmMax   := TRUE;
   END_REGION
   REGION X_Axis_Temperature_PTC
       "DB_AnalogInputDataPLC".X_Axis_Temperature_PTC.EnableAlarmMin   := FALSE;
       "DB_AnalogInputDataPLC".X_Axis_Temperature_PTC.EnableWarningMin := FALSE;
       "DB_AnalogInputDataPLC".X_Axis_Temperature_PTC.EnableWarningMax := FALSE;
       "DB_AnalogInputDataPLC".X_Axis_Temperature_PTC.EnableAlarmMax   := FALSE;
   END_REGION

   REGION Y_Axis_Temperature_PTC
       "DB_AnalogInputDataPLC".Y_Axis_Temperature_PTC.EnableAlarmMin   := FALSE;
       "DB_AnalogInputDataPLC".Y_Axis_Temperature_PTC.EnableWarningMin := FALSE;
       "DB_AnalogInputDataPLC".Y_Axis_Temperature_PTC.EnableWarningMax := FALSE;
       "DB_AnalogInputDataPLC".Y_Axis_Temperature_PTC.EnableAlarmMax   := FALSE;
   END_REGION

   REGION Nozzle_Overpressure
       "DB_AnalogInputDataPLC".Nozzle_Overpressure.EnableAlarmMin   := TRUE;
       "DB_AnalogInputDataPLC".Nozzle_Overpressure.EnableWarningMin := TRUE;
       "DB_AnalogInputDataPLC".Nozzle_Overpressure.EnableWarningMax := TRUE;
       "DB_AnalogInputDataPLC".Nozzle_Overpressure.EnableAlarmMax   := TRUE;
   END_REGION

   REGION Optical_Path_Overpressure
       "DB_AnalogInputDataPLC".Optical_Path_Overpressure.EnableAlarmMin   := TRUE;
       "DB_AnalogInputDataPLC".Optical_Path_Overpressure.EnableWarningMin := TRUE;
       "DB_AnalogInputDataPLC".Optical_Path_Overpressure.EnableWarningMax := TRUE;
       "DB_AnalogInputDataPLC".Optical_Path_Overpressure.EnableAlarmMax   := TRUE;
   END_REGION

   REGION Laser_Head_Overpressure
       "DB_AnalogInputDataPLC".Laser_Head_Overpressure.EnableAlarmMin   := TRUE;
       "DB_AnalogInputDataPLC".Laser_Head_Overpressure.EnableWarningMin := TRUE;
       "DB_AnalogInputDataPLC".Laser_Head_Overpressure.EnableWarningMax := TRUE;
       "DB_AnalogInputDataPLC".Laser_Head_Overpressure.EnableAlarmMax   := TRUE;
   END_REGION

   REGION ZL_Axis_Overpressure
       "DB_AnalogInputDataPLC".ZL_Axis_Overpressure.EnableAlarmMin   := TRUE;
       "DB_AnalogInputDataPLC".ZL_Axis_Overpressure.EnableWarningMin := TRUE;
       "DB_AnalogInputDataPLC".ZL_Axis_Overpressure.EnableWarningMax := TRUE;
       "DB_AnalogInputDataPLC".ZL_Axis_Overpressure.EnableAlarmMax   := TRUE;
   END_REGION

   REGION XY_Axis_Overpressure
       "DB_AnalogInputDataPLC".XY_Axis_Overpressure.EnableAlarmMin   := TRUE;
       "DB_AnalogInputDataPLC".XY_Axis_Overpressure.EnableWarningMin := TRUE;
       "DB_AnalogInputDataPLC".XY_Axis_Overpressure.EnableWarningMax := TRUE;
       "DB_AnalogInputDataPLC".XY_Axis_Overpressure.EnableAlarmMax   := TRUE;
   END_REGION

   REGION Left_Aspiration
       "DB_AnalogInputDataPLC".Left_Aspiration.EnableAlarmMin   := TRUE;
       "DB_AnalogInputDataPLC".Left_Aspiration.EnableWarningMin := TRUE;
       "DB_AnalogInputDataPLC".Left_Aspiration.EnableWarningMax := TRUE;
       "DB_AnalogInputDataPLC".Left_Aspiration.EnableAlarmMax   := TRUE;
   END_REGION

   REGION Right_Aspiration
       "DB_AnalogInputDataPLC".Right_Aspiration.EnableAlarmMin   := TRUE;
       "DB_AnalogInputDataPLC".Right_Aspiration.EnableWarningMin := TRUE;
       "DB_AnalogInputDataPLC".Right_Aspiration.EnableWarningMax := TRUE;
       "DB_AnalogInputDataPLC".Right_Aspiration.EnableAlarmMax   := TRUE;
   END_REGION

   REGION Clim_Temperature
       "DB_AnalogInputDataPLC".Clim_Temperature.EnableAlarmMin   := FALSE;
       "DB_AnalogInputDataPLC".Clim_Temperature.EnableWarningMin := FALSE;
       "DB_AnalogInputDataPLC".Clim_Temperature.EnableWarningMax := FALSE;
       "DB_AnalogInputDataPLC".Clim_Temperature.EnableAlarmMax   := FALSE;
   END_REGION

   REGION Sensor_Controller_Station1
       "DB_AnalogInputDataPLC".Sensor_Controller_Station1.EnableAlarmMin   := FALSE;
       "DB_AnalogInputDataPLC".Sensor_Controller_Station1.EnableWarningMin := FALSE;
       "DB_AnalogInputDataPLC".Sensor_Controller_Station1.EnableWarningMax := FALSE;
       "DB_AnalogInputDataPLC".Sensor_Controller_Station1.EnableAlarmMax   := FALSE;
   END_REGION

   REGION Cabinet_Temperature
       "DB_AnalogInputDataPLC".Cabinet_Temperature.EnableAlarmMin   := FALSE;
       "DB_AnalogInputDataPLC".Cabinet_Temperature.EnableWarningMin := FALSE;
       "DB_AnalogInputDataPLC".Cabinet_Temperature.EnableWarningMax := FALSE;
       "DB_AnalogInputDataPLC".Cabinet_Temperature.EnableAlarmMax   := FALSE;
   END_REGION
END_FUNCTION

FUNCTION_BLOCK "FB_Nouveau_1"
{ S7_Optimized_Access := 'TRUE' }
VERSION : 0.1
   VAR 
      "#sExtLoadUnloadTimer1" {InstructionName := 'TON_TIME'; LibVersion := '1.0'; S7_SetPoint := 'False'} : TON_TIME;
      "#sExtLoadUnloadTimer2" {InstructionName := 'TON_TIME'; LibVersion := '1.0'} : TON_TIME;
   END_VAR


BEGIN
	REGION Ext Load/Unload Time
	    // Necessaire pour Dry Run
	    // #sExtLoadUnloadTimer1(IN := "DB_LoaderShuttle1".sExtLoadUnload.sCurrent_Step_NB = 50
	    //                       OR "DB_LoaderShuttle1".sExtLoadUnload.sCurrent_Step_NB = 80
	    //                       OR "DB_LoaderShuttle1".sExtLoadUnload.sCurrent_Step_NB = 110,
	    //                       PT := t#3s);
	    // "DB_SonplasMain".sSonplasLoader.iPartInShuttle1Finished := #sExtLoadUnloadTimer1.Q;
	    
	    // #sExtLoadUnloadTimer2(IN := "DB_LoaderShuttle2".sExtLoadUnload.sCurrent_Step_NB = 50
	    //                       OR "DB_LoaderShuttle2".sExtLoadUnload.sCurrent_Step_NB = 80
	    //                       OR "DB_LoaderShuttle2".sExtLoadUnload.sCurrent_Step_NB = 110,
	    //                       PT := t#3s);
	    // "DB_SonplasMain".sSonplasLoader.iPartInShuttle2Finished := #sExtLoadUnloadTimer2.Q;
	END_REGION
END_FUNCTION_BLOCK

FUNCTION_BLOCK "FB_Simulation_1"
{ S7_Optimized_Access := 'TRUE' }
VERSION : 0.1
   VAR 
      sExtLoadUnloadTimer1 {InstructionName := 'TON_TIME'; LibVersion := '1.0'; S7_SetPoint := 'False'} : TON_TIME;
      sExtLoadUnloadTimer2 {InstructionName := 'TON_TIME'; LibVersion := '1.0'} : TON_TIME;
      sBwLoadUnloadTimer1 {InstructionName := 'TON_TIME'; LibVersion := '1.0'} : TON_TIME;
      sBwLoadUnloadTimer2 {InstructionName := 'TON_TIME'; LibVersion := '1.0'} : TON_TIME;
      sTON_UndrilledGripperFull {InstructionName := 'TON_TIME'; LibVersion := '1.0'} : TON_TIME;
      sTON_UndrilledFixture {InstructionName := 'TON_TIME'; LibVersion := '1.0'} : TON_TIME;
      sTON_DrilledFixture {InstructionName := 'TON_TIME'; LibVersion := '1.0'} : TON_TIME;
      sTON_ResetBit {InstructionName := 'TON_TIME'; LibVersion := '1.0'} : TON_TIME;
      sSeqRun { S7_SetPoint := 'True'} : Bool;
      sTON_CloseDrilledGripper_1 {InstructionName := 'TON_TIME'; LibVersion := '1.0'} : TON_TIME;
      sTONCloseFixture {InstructionName := 'TON_TIME'; LibVersion := '1.0'} : TON_TIME;
      sTONOpenFixture {InstructionName := 'TON_TIME'; LibVersion := '1.0'} : TON_TIME;
      sTONOpenFixture1 {InstructionName := 'TON_TIME'; LibVersion := '1.0'} : TON_TIME;
      sTON_CloseDrilledGripper {InstructionName := 'TON_TIME'; LibVersion := '1.0'} : TON_TIME;
      sTON_WorkinProgress {InstructionName := 'TON_TIME'; LibVersion := '1.0'} : TON_TIME;
      sTON_OpenUndrilledGripper {InstructionName := 'TON_TIME'; LibVersion := '1.0'} : TON_TIME;
      sRT_NC_Mode {InstructionName := 'R_TRIG'; LibVersion := '1.0'} : R_TRIG;
      sStep { S7_SetPoint := 'True'} : Array[0..15] of Bool;
      sRT_DrillingFinished {InstructionName := 'R_TRIG'; LibVersion := '1.0'; S7_SetPoint := 'False'} : R_TRIG;
      "sTON_No MCodes" {InstructionName := 'TON_TIME'; LibVersion := '1.0'} : TON_TIME;
      sRT_TONMCodes {InstructionName := 'R_TRIG'; LibVersion := '1.0'} : R_TRIG;
      sRT_FIXLoading {InstructionName := 'R_TRIG'; LibVersion := '1.0'} : R_TRIG;
      sRT_FIXblowing {InstructionName := 'R_TRIG'; LibVersion := '1.0'} : R_TRIG;
      sRT_MemoLoaderStart {InstructionName := 'R_TRIG'; LibVersion := '1.0'} : R_TRIG;
      sRT_Sh1_ExtLoadUnloadDone {InstructionName := 'R_TRIG'; LibVersion := '1.0'} : R_TRIG;
      sRT_Sh2_ExtLoadUnloadDone {InstructionName := 'R_TRIG'; LibVersion := '1.0'} : R_TRIG;
   END_VAR


BEGIN
	REGION Ext Load/Unload Time
	    // Necessaire pour Dry Run
	    #sExtLoadUnloadTimer1(IN:= "DB_LoaderShuttle1".sExtLoadUnload.sCurrent_Step_NB = 50
	                          OR "DB_LoaderShuttle1".sExtLoadUnload.sCurrent_Step_NB = 80
	                          OR "DB_LoaderShuttle1".sExtLoadUnload.sCurrent_Step_NB = 110,
	                          PT:= t#3s);
	   "DB_SonplasMain".sSonplasLoader.iPartInShuttle1Finished := #sExtLoadUnloadTimer1.Q;
	   
	   #sExtLoadUnloadTimer2(IN :=  "DB_LoaderShuttle2".sExtLoadUnload.sCurrent_Step_NB = 50
	                         OR "DB_LoaderShuttle2".sExtLoadUnload.sCurrent_Step_NB = 80
	                         OR "DB_LoaderShuttle2".sExtLoadUnload.sCurrent_Step_NB = 110,
	                         PT := t#3s);
	   "DB_SonplasMain".sSonplasLoader.iPartInShuttle2Finished := #sExtLoadUnloadTimer2.Q;
	END_REGION
	
	REGION Bw Load/Unload Time
	    // Necessaire pour Dry Run
	    #sBwLoadUnloadTimer1(IN := "DB_LoaderShuttle1".sBwLoadUnload.sCurrent_Step_NB = 50
	                         OR "DB_LoaderShuttle1".sBwLoadUnload.sCurrent_Step_NB = 150,
	                         PT := t#2s);
	    
	    #sBwLoadUnloadTimer2(IN := "DB_LoaderShuttle2".sBwLoadUnload.sCurrent_Step_NB = 50
	                         OR "DB_LoaderShuttle2".sBwLoadUnload.sCurrent_Step_NB = 150,
	                         PT := t#2s);
	  //  "DB_BwLoader".sBwCommunication.oLoadJobDone := #sBwLoadUnloadTimer1.Q OR #sBwLoadUnloadTimer2.Q;
	  //  "DB_BwLoader".sBwCommunication.oUnloadJobDone := #sBwLoadUnloadTimer1.Q OR #sBwLoadUnloadTimer2.Q;
	END_REGION
	   
	REGION Part Position  
	   // Necessaire pour Dry Run
	    IF ("DB_LoaderShuttle1".sControlIn.sInterface.SequenceRun OR "DB_LoaderShuttle2".sControlIn.sInterface.SequenceRun) AND NOT "DB_WAF".CtrlInEnable THEN
	       IF "DB_WorkingModes".sFilling THEN
	           "DB_DigitalInputsBW_Station".sUndrilledPartCtrl.sSWStatus := TRUE;
	           "DB_DigitalInputsBW_Station".sDrilledPartCtrl.sSWStatus := FALSE;
	       ELSIF "DB_WorkingModes".sNormal THEN
	           "DB_DigitalInputsBW_Station".sUndrilledPartCtrl.sSWStatus := TRUE;
	           "DB_DigitalInputsBW_Station".sDrilledPartCtrl.sSWStatus := FALSE;
	       ELSIF "DB_WorkingModes".sEmptying THEN
	           "DB_DigitalInputsBW_Station".sUndrilledPartCtrl.sSWStatus := FALSE;
	           "DB_DigitalInputsBW_Station".sDrilledPartCtrl.sSWStatus := FALSE;
	       END_IF;
	   END_IF;
	   
	   IF ("DB_LoaderShuttle1".sControlOut.sInterface.SequenceRun OR "DB_LoaderShuttle2".sControlOut.sInterface.SequenceRun) AND NOT "DB_WAF".CtrlOutEnable THEN
	       IF "DB_WorkingModes".sFilling THEN
	           "DB_DigitalInputsBW_Station".sUndrilledPartCtrl.sSWStatus := FALSE;
	           "DB_DigitalInputsBW_Station".sDrilledPartCtrl.sSWStatus := FALSE;
	       ELSIF "DB_WorkingModes".sNormal THEN
	           "DB_DigitalInputsBW_Station".sUndrilledPartCtrl.sSWStatus := FALSE;
	           "DB_DigitalInputsBW_Station".sDrilledPartCtrl.sSWStatus := TRUE;
	       ELSIF "DB_WorkingModes".sEmptying THEN
	           "DB_DigitalInputsBW_Station".sUndrilledPartCtrl.sSWStatus := FALSE;
	           "DB_DigitalInputsBW_Station".sDrilledPartCtrl.sSWStatus := TRUE;
	       END_IF;
	   END_IF;
	 END_REGION
	
	 REGION BW Position
	     // Necessaire pour Dry Run
	     IF NOT "DB_WAF".CtrlBwEnable THEN
	         IF "DB_WorkingModes".sNormal THEN
	             "DB_DigitalInputsBW_Station".sBwCtrl.sSWStatus := TRUE;
	         ELSIF "DB_WorkingModes".sEmptying THEN
	             // "DB_DigitalInputsBW_Station".sBwCtrl.sSWStatus := FALSE;
	             "DB_DigitalInputsBW_Station".sBwCtrl.sSWStatus := "DB_PartManagement".sPosition.sShuttle1.Undrilled.Presence.Part
	             OR "DB_PartManagement".sPosition.sShuttle1.Undrilled.Presence.Part;
	         ELSIF "DB_WorkingModes".sFilling THEN
	             "DB_DigitalInputsBW_Station".sBwCtrl.sSWStatus := TRUE;
	         END_IF;
	     END_IF;
	     END_REGION
	
	REGION Drilling Finished
	   // Necessaire pour Dry Run
	    #sRT_DrillingFinished(CLK := "DB_PartManagement".sPosition.sFixture.Undrilled.Presence.Part AND "DB_PartManagement".sPosition.sFixture.Undrilled.Presence.BW);
	    "DB_PartManagement".sPosition.iDrilling_Finished := #sRT_DrillingFinished.Q;
	END_REGION
	
	REGION Interlock
	   "DB_WAF".Sonplas.OperateInOutCollision := TRUE;
	   "DB_WAF".BwLoader.Safe := TRUE;
	   "DB_WAF".bSpy[9] := "DB_WAF".bSpy[9];
// test modif depuis repo Git
	END_REGION
	
	REGION Ext Loader
	    "DB_LoaderOptions".ExtLoadUnload.Disabled := TRUE;
	    
	    #sRT_Sh1_ExtLoadUnloadDone(CLK := "DB_LoaderShuttle1".sExtLoadUnload.sInterface.JobDone);
	    #sRT_Sh2_ExtLoadUnloadDone(CLK := "DB_LoaderShuttle2".sExtLoadUnload.sInterface.JobDone);
	    
	    IF #sRT_Sh1_ExtLoadUnloadDone.Q THEN
	        "DB_SonplasMain".sSonplasLoader.iPartInDMC_CodeShuttle1[0] := "DB_SonplasMain".sSonplasLoader.iPartInDMC_CodeShuttle1[0] + 1;
	        IF "DB_SonplasMain".sSonplasLoader.iPartInDMC_CodeShuttle1[0] > 99 THEN
	            "DB_SonplasMain".sSonplasLoader.iPartInDMC_CodeShuttle1[0] := 0;
	        END_IF;
	    END_IF;
	    
	    IF #sRT_Sh2_ExtLoadUnloadDone.Q THEN
	        "DB_SonplasMain".sSonplasLoader.iPartInDMC_CodeShuttle2[0] := "DB_SonplasMain".sSonplasLoader.iPartInDMC_CodeShuttle2[0] + 1;
	        IF "DB_SonplasMain".sSonplasLoader.iPartInDMC_CodeShuttle2[0] > 99 THEN
	            "DB_SonplasMain".sSonplasLoader.iPartInDMC_CodeShuttle2[0] := 0;
	        END_IF;
	    END_IF;
	END_REGION
	    
	// REGION Shuttle Enable
	//     "DB_HMISetting".Shuttle1Enable := TRUE;
	//     "DB_HMISetting".Shuttle2Enable := TRUE;
	// END_REGION
	   
	REGION Misc
	       "DB_WorkingModes".sDryRun := FALSE;
	END_REGION
	
	REGION Reset Part Position
	    IF "DB_WAF".ResetPartPosition THEN
	        "DB_PartManagement".sPosition.sShuttle1.Undrilled.Presence.Part := FALSE;
	        "DB_PartManagement".sPosition.sShuttle1.Undrilled.Presence.BW := FALSE;
	        "DB_PartManagement".sPosition.sShuttle1.Drilled.Presence.Part := FALSE;
	        "DB_PartManagement".sPosition.sShuttle1.Drilled.Presence.BW := FALSE;
	        
	        "DB_PartManagement".sPosition.sShuttle2.Undrilled.Presence.Part := FALSE;
	        "DB_PartManagement".sPosition.sShuttle2.Undrilled.Presence.BW := FALSE;
	        "DB_PartManagement".sPosition.sShuttle2.Drilled.Presence.Part := FALSE;
	        "DB_PartManagement".sPosition.sShuttle2.Drilled.Presence.BW := FALSE;
	        
	        "DB_PartManagement".sPosition.sGripper.Undrilled.Presence.Part := FALSE;
	        "DB_PartManagement".sPosition.sGripper.Undrilled.Presence.BW := FALSE;
	        "DB_PartManagement".sPosition.sGripper.Drilled.Presence.Part := FALSE;
	        "DB_PartManagement".sPosition.sGripper.Drilled.Presence.BW := FALSE;
	        
	        "DB_PartManagement".sPosition.sFixture.Undrilled.Presence.Part := FALSE;
	        "DB_PartManagement".sPosition.sFixture.Undrilled.Presence.BW := FALSE;
	        "DB_PartManagement".sPosition.sFixture.Drilled.Presence.Part := FALSE;
	        "DB_PartManagement".sPosition.sFixture.Drilled.Presence.BW := FALSE;
	        
	        "DB_WAF".ResetPartPosition := FALSE;
	        "DB_WAF".NewTag_2 := FALSE;
	    END_IF;
	END_REGION
END_FUNCTION_BLOCK

DATA_BLOCK "DB_HMI_PLC_Pos"   // DB135
// stored: InstanceOfName FB_HMI_PLC_Pos, InstanceOfType FB
"FB_HMI_PLC_Pos"
BEGIN
END_DATA_BLOCK

DATA_BLOCK "DB_Simulation"   // DB99
// stored: InstanceOfName FB_Simulation, InstanceOfType FB
"FB_Simulation"
BEGIN
END_DATA_BLOCK

DATA_BLOCK "DB_FeedOverride"   // DB116
// stored: InstanceOfName FB_FeedOverride, InstanceOfType FB
"FB_FeedOverride"
BEGIN
END_DATA_BLOCK

DATA_BLOCK "DB_Impulsion"   // DB84
// stored: InstanceOfName FB_Impulsion, InstanceOfType FB
"FB_Impulsion"
BEGIN
END_DATA_BLOCK

DATA_BLOCK "DB_ReadDateAndTime"   // DB9
// stored: InstanceOfName FB_ReadDateAndTime, InstanceOfType FB
"FB_ReadDateAndTime"
BEGIN
END_DATA_BLOCK

DATA_BLOCK "DB_CommPLC_ISO"   // DB1100
// stored: AutoNumber false, InstanceOfName FB_CommPLC_ISO, InstanceOfType FB
"FB_CommPLC_ISO"
BEGIN
END_DATA_BLOCK

DATA_BLOCK "DB_MiscPLC_IHM_ISO"   // DB97
// stored: InstanceOfName FB_MiscPLC_IHM_ISO, InstanceOfType FB
"FB_MiscPLC_IHM_ISO"
BEGIN
END_DATA_BLOCK

DATA_BLOCK "Main_Safety_RTG1_DB"   // DB62, F_DB
NAME : FUSI
// stored: InstanceOfName Main_Safety_RTG1, InstanceOfType FB
"Main_Safety_RTG1"
BEGIN
END_DATA_BLOCK

DATA_BLOCK "DBI_GUD_VERSION"   // DB1201
// stored: AutoNumber false, InstanceOfName FB_ReadWrite_GUDs, InstanceOfType FB
"FB_ReadWrite_GUDs"
BEGIN
END_DATA_BLOCK

DATA_BLOCK "DB_ExtraMissingPart"   // DB113
// stored: InstanceOfName FB_ExtraMissingPart, InstanceOfType FB
"FB_ExtraMissingPart"
BEGIN
END_DATA_BLOCK

DATA_BLOCK "DB_LoaderAxis"   // DB206
// stored: AutoNumber false, InstanceOfName FB_LoaderAxis, InstanceOfType FB
"FB_LoaderAxis"
BEGIN
END_DATA_BLOCK

DATA_BLOCK "DB_LoaderMain"   // DB203
// stored: AutoNumber false, InstanceOfName FB_LoaderMain, InstanceOfType FB
"FB_LoaderMain"
BEGIN
END_DATA_BLOCK

DATA_BLOCK "DB_LoaderShuttle1"   // DB204
// stored: AutoNumber false, InstanceOfName FB_LoaderShuttle1, InstanceOfType FB
"FB_LoaderShuttle1"
BEGIN
END_DATA_BLOCK

DATA_BLOCK "DB_LoaderShuttle2"   // DB205
// stored: AutoNumber false, InstanceOfName FB_LoaderShuttle2, InstanceOfType FB
"FB_LoaderShuttle2"
BEGIN
END_DATA_BLOCK

DATA_BLOCK "DB_PartManagement"   // DB87
// stored: InstanceOfName FB_PartManagement, InstanceOfType FB
"FB_PartManagement"
BEGIN
END_DATA_BLOCK

DATA_BLOCK "DB_PrioSequence"   // DB114
// stored: InstanceOfName FB_PrioSequence, InstanceOfType FB
"FB_PrioSequence"
BEGIN
END_DATA_BLOCK

DATA_BLOCK "DB_LoaderFixture"   // DB106
// stored: InstanceOfName FB_LoaderFixture, InstanceOfType FB
"FB_LoaderFixture"
BEGIN
END_DATA_BLOCK

DATA_BLOCK "DB_LoaderFixtureMain"   // DB4
// stored: InstanceOfName FB_LoaderFixtureMain, InstanceOfType FB
"FB_LoaderFixtureMain"
BEGIN
END_DATA_BLOCK

DATA_BLOCK "DB_Alarms"   // DB300
// stored: AutoNumber false, InstanceOfName FB_Alarms, InstanceOfType FB
"FB_Alarms"
BEGIN
END_DATA_BLOCK

DATA_BLOCK "DB_Msg"   // DB13
// stored: InstanceOfName FB_Msg, InstanceOfType FB
"FB_Msg"
BEGIN
END_DATA_BLOCK

DATA_BLOCK "DB_Tracability"   // DB94
// stored: InstanceOfName FB_Tracability, InstanceOfType FB
"FB_Tracability"
BEGIN
END_DATA_BLOCK

DATA_BLOCK "DB_DataFromSafety"   // DB122
{ S7_Optimized_Access := 'TRUE' }
// stored: AutoNumber false, InstanceOfName DT_DataFromSafety, InstanceOfType UDT
"DT_DataFromSafety"
BEGIN
END_DATA_BLOCK

DATA_BLOCK "DB_DataToSafety"   // DB120
{ S7_Optimized_Access := 'TRUE' }
// stored: AutoNumber false, InstanceOfName DT_DataToSafety, InstanceOfType UDT
"DT_DataToSafety"
BEGIN
END_DATA_BLOCK

DATA_BLOCK "F-DB_DataFromSafety"   // DB123, F_DB
{ S7_Optimized_Access := 'TRUE' }
// stored: AutoNumber false, InstanceOfName DT_DataFromSafety, InstanceOfType UDT
"DT_DataFromSafety"
BEGIN
END_DATA_BLOCK

DATA_BLOCK "F-DB_DataToSafety"   // DB121, F_DB
{ S7_Optimized_Access := 'TRUE' }
// stored: AutoNumber false, InstanceOfName DT_DataToSafety, InstanceOfType UDT
"DT_DataToSafety"
BEGIN
END_DATA_BLOCK

DATA_BLOCK "F-DB_Axis"   // DB130, F_DB
// stored: AutoNumber false, InstanceOfName F-FB_Axis, InstanceOfType FB
"F-FB_Axis"
BEGIN
END_DATA_BLOCK

DATA_BLOCK "F-DB_Laser"   // DB140, F_DB
// stored: AutoNumber false, InstanceOfName F-FB_Laser, InstanceOfType FB
"F-FB_Laser"
BEGIN
END_DATA_BLOCK

DATA_BLOCK "DB_Alarms_Safety"   // DB150
// stored: AutoNumber false, InstanceOfName FB_Alarms_Safety, InstanceOfType FB
"FB_Alarms_Safety"
BEGIN
END_DATA_BLOCK

DATA_BLOCK "DB_SonplasMain"   // DB88
// stored: InstanceOfName FB_SonplasMain, InstanceOfType FB
"FB_SonplasMain"
BEGIN
   sSonplasLoader.iPartInDMC_CodeShuttle1[0] := 16#0;
END_DATA_BLOCK

DATA_BLOCK "DB_HmiKeyboardSignals"   // DB90
// stored: InstanceOfName FB_HmiKeyboardSignals, InstanceOfType FB
"FB_HmiKeyboardSignals"
BEGIN
END_DATA_BLOCK

DATA_BLOCK "DB_OPC_AxisManagement"   // DB105
// stored: InstanceOfName FB_OPC_AxisManagement, InstanceOfType FB
"FB_OPC_AxisManagement"
BEGIN
END_DATA_BLOCK

DATA_BLOCK "DB_OPC_State"   // DB112
// stored: InstanceOfName FB_OPC_State, InstanceOfType FB
"FB_OPC_State"
BEGIN
END_DATA_BLOCK

DATA_BLOCK "DB_BwLoader"   // DB108
// stored: InstanceOfName FB_BwLoader, InstanceOfType FB
"FB_BwLoader"
BEGIN
END_DATA_BLOCK

DATA_BLOCK "DB_RealTime"   // DB107
// stored: InstanceOfName FB_RealTime, InstanceOfType FB
"FB_RealTime"
BEGIN
END_DATA_BLOCK

DATA_BLOCK "DB_Components"   // DB119
// stored: InstanceOfName FB_Components, InstanceOfType FB
"FB_Components"
BEGIN
END_DATA_BLOCK

DATA_BLOCK "DB_Parameters"   // DB109
// stored: InstanceOfName FB_Parameters, InstanceOfType FB
"FB_Parameters"
BEGIN
END_DATA_BLOCK

DATA_BLOCK "DB_Part_Data"   // DB131
// stored: InstanceOfName FB_Part_Data, InstanceOfType FB
"FB_Part_Data"
BEGIN
END_DATA_BLOCK

DATA_BLOCK "DB_Scanner"   // DB128
// stored: InstanceOfName FB_Scanner, InstanceOfType FB
"FB_Scanner"
BEGIN
END_DATA_BLOCK

DATA_BLOCK "DB_ScannerComm"   // DB126
// stored: InstanceOfName FB_ScannerComm, InstanceOfType FB
"FB_ScannerComm"
BEGIN
END_DATA_BLOCK

DATA_BLOCK "LBP_ReadVar_DB_R_Param"   // DB129
// stored: InstanceOfName LBP_ReadVar, InstanceOfType FB
"LBP_ReadVar"
   // VAR_INPUT
   //    Req : Bool;
   //    NumVar : Int;
   //    Addr1 : Variant;
   //    Unit1 : Byte;
   //    Column1 : Word;
   //    Line1 : Word;
   //    Addr2 : Variant;
   //    Unit2 : Byte;
   //    Column2 : Word;
   //    Line2 : Word;
   //    Addr3 : Variant;
   //    Unit3 : Byte;
   //    Column3 : Word;
   //    Line3 : Word;
   //    Addr4 : Variant;
   //    Unit4 : Byte;
   //    Column4 : Word;
   //    Line4 : Word;
   //    Addr5 : Variant;
   //    Unit5 : Byte;
   //    Column5 : Word;
   //    Line5 : Word;
   //    Addr6 : Variant;
   //    Unit6 : Byte;
   //    Column6 : Word;
   //    Line6 : Word;
   //    Addr7 : Variant;
   //    Unit7 : Byte;
   //    Column7 : Word;
   //    Line7 : Word;
   //    Addr8 : Variant;
   //    Unit8 : Byte;
   //    Column8 : Word;
   //    Line8 : Word;
   // END_VAR
   // VAR_OUTPUT
   //    Error : Bool;
   //    NDR : Bool;
   //    State : Word;
   // END_VAR
   // VAR_IN_OUT
   //    RD1 : Variant;
   //    RD2 : Variant;
   //    RD3 : Variant;
   //    RD4 : Variant;
   //    RD5 : Variant;
   //    RD6 : Variant;
   //    RD7 : Variant;
   //    RD8 : Variant;
   // END_VAR
   // VAR
   //    ident : Byte;
   //    regist : Bool;
   //    flanke : Bool;
   //    progtest : Bool;
   //    err_cls_cod : Word;
   //    err_stat : Word;
   //    s_fifoRef : UInt;
   //    s_Reserved1 : Word;
   //    s_Reserved2 : DWord;
   //    s_Reserved3 : DWord;
   // END_VAR
BEGIN
END_DATA_BLOCK

DATA_BLOCK "DB_Recipe"   // DB133
// stored: InstanceOfName FB_Recipe, InstanceOfType FB
"FB_Recipe"
BEGIN
END_DATA_BLOCK

DATA_BLOCK "DB_GestionSafetyGate"   // DB202
// stored: AutoNumber false, InstanceOfName FB_GestionSafetyGate, InstanceOfType FB
"FB_GestionSafetyGate"
BEGIN
END_DATA_BLOCK

DATA_BLOCK "DB_GestionGripper"   // DB64
// stored: InstanceOfName FB_GestionGripper, InstanceOfType FB
"FB_GestionGripper"
BEGIN
END_DATA_BLOCK

DATA_BLOCK "DB_GestionFixture"   // DB89
// stored: InstanceOfName FB_GestionFixture, InstanceOfType FB
"FB_GestionFixture"
BEGIN
END_DATA_BLOCK

DATA_BLOCK "DB_GestionWorkingModes"   // DB132
// stored: InstanceOfName FB_GestionWorkingModes, InstanceOfType FB
"FB_GestionWorkingModes"
BEGIN
END_DATA_BLOCK

DATA_BLOCK "DB_WorkingModes"   // DB100
// stored: InstanceOfName FB_WorkingModes, InstanceOfType FB
"FB_WorkingModes"
BEGIN
END_DATA_BLOCK

DATA_BLOCK "DB_CycleStartStop"   // DB81
// stored: InstanceOfName FB_CycleStartStop, InstanceOfType FB
"FB_CycleStartStop"
BEGIN
END_DATA_BLOCK

DATA_BLOCK "DB_DecodChannels"   // DB405
{ DB_Accessible_From_OPC_UA := 'FALSE' }
AUTHOR : BAJ
// stored: AutoNumber false, DBAccessibleFromOPCUA false, DBAccessibleFromWebserver false, InstanceOfName FB_DecodChannels, InstanceOfType FB
"FB_DecodChannels"
BEGIN
END_DATA_BLOCK

DATA_BLOCK "DB_Axis"   // DB410
// stored: AutoNumber false, InstanceOfName FB_Axis, InstanceOfType FB
"FB_Axis"
BEGIN
END_DATA_BLOCK

DATA_BLOCK "DB_AxisPosition"   // DB411
// stored: AutoNumber false, InstanceOfName FB_AxisPosition, InstanceOfType FB
"FB_AxisPosition"
BEGIN
END_DATA_BLOCK

DATA_BLOCK "DB_MCPManagement"   // DB425
// stored: AutoNumber false, InstanceOfName FB_MCPManagement, InstanceOfType FB
"FB_MCPManagement"
BEGIN
END_DATA_BLOCK

DATA_BLOCK "DB_McpKeyboardSignals"   // DB421
// stored: AutoNumber false, InstanceOfName FB_McpKeyboardSignals, InstanceOfType FB
"FB_McpKeyboardSignals"
BEGIN
END_DATA_BLOCK

DATA_BLOCK "DB_LaserAirProcess"   // DB432
// stored: AutoNumber false, InstanceOfName FB_LaserAirProcess, InstanceOfType FB
"FB_LaserAirProcess"
BEGIN
END_DATA_BLOCK

DATA_BLOCK "DB_LaserMeasureZoneSwitch"   // DB91
// stored: InstanceOfName FB_LaserMeasureZoneSwitch, InstanceOfType FB
"FB_LaserMeasureZoneSwitch"
BEGIN
END_DATA_BLOCK

DATA_BLOCK "DB_LaserOperation"   // DB431
// stored: AutoNumber false, InstanceOfName FB_LaserOperation, InstanceOfType FB
"FB_LaserOperation"
BEGIN
END_DATA_BLOCK

DATA_BLOCK "DB_Powermeter"   // DB433
// stored: AutoNumber false, InstanceOfName FB_Powermeter, InstanceOfType FB
"FB_Powermeter"
BEGIN
END_DATA_BLOCK

DATA_BLOCK "DB_PowermeterMeasures"   // DB434
TITLE = DB_MEAS_POWER_METER
{ S7_Optimized_Access := 'TRUE' }
AUTHOR : SAN
// Measures of power metter
// stored: AutoNumber false, InstanceOfName UDT_PowermeterMeasure, InstanceOfType UDT
"UDT_PowermeterMeasure"
BEGIN
END_DATA_BLOCK

DATA_BLOCK "DB_Pressures"   // DB440
// stored: InstanceOfName FB_Pressures, InstanceOfType FB
"FB_Pressures"
BEGIN
END_DATA_BLOCK

DATA_BLOCK "DB_Vacuums"   // DB441
// stored: AutoNumber false, InstanceOfName FB_Vacuums, InstanceOfType FB
"FB_Vacuums"
BEGIN
END_DATA_BLOCK

DATA_BLOCK "DB_Cognex"   // DB1255
// stored: AutoNumber false, InstanceOfName FB_Cognex, InstanceOfType FB
"FB_Cognex"
BEGIN
END_DATA_BLOCK

DATA_BLOCK "DB_Machineshutdown_UPS"   // DB461
// stored: AutoNumber false, InstanceOfName FB_Machineshutdown_UPS, InstanceOfType FB
"FB_Machineshutdown_UPS"
BEGIN
END_DATA_BLOCK

DATA_BLOCK "DB_PowerOn"   // DB462
// stored: AutoNumber false, InstanceOfName FB_PowerOn, InstanceOfType FB
"FB_PowerOn"
BEGIN
END_DATA_BLOCK

DATA_BLOCK "DB_Maintenances"   // DB20
// stored: InstanceOfName FB_Maintenances, InstanceOfType FB
"FB_Maintenances"
BEGIN
   sCheckMachine.sElement.RunTimeSec := 0.0;
   sCheckMachine.sElement.WarningThreshold := 160;
   sCheckMachine.sElement.AlarmThreshold := 200;
   sReplaceAirConditioningFilter.sElement.RunTimeSec := 0.0;
   sReplaceAirConditioningFilter.sElement.WarningThreshold := 800;
   sReplaceAirConditioningFilter.sElement.AlarmThreshold := 1000;
   sMachineCooling_ReplaceWaterFilter.sElement.WarningThreshold := 800;
   sMachineCooling_ReplaceWaterFilter.sElement.AlarmThreshold := 1000;
   sTermotekChiller_ChangeFilterAndWater.sElement.WarningThreshold := 1600;
   sTermotekChiller_ChangeFilterAndWater.sElement.AlarmThreshold := 2000;
   sCheckSafetySystem.sElement.WarningThreshold := 1600;
   sCheckSafetySystem.sElement.AlarmThreshold := 2000;
   sReplaceTipShellPeekGripper.sElement.WarningThreshold := 1600;
   sReplaceTipShellPeekGripper.sElement.AlarmThreshold := 2000;
   sReplaceFiltersVacuumLoadingUnloading.sElement.WarningThreshold := 2400;
   sReplaceFiltersVacuumLoadingUnloading.sElement.AlarmThreshold := 3000;
   sReplaceFiltersVacuumGenerator.sElement.WarningThreshold := 2400;
   sReplaceFiltersVacuumGenerator.sElement.AlarmThreshold := 3000;
   sReplaceFilterAirDryer.sElement.WarningThreshold := 3200;
   sReplaceFilterAirDryer.sElement.AlarmThreshold := 4000;
   sReplace5umFilter.sElement.WarningThreshold := 3200;
   sReplace5umFilter.sElement.AlarmThreshold := 4000;
   sReplace01umFilter.sElement.WarningThreshold := 3200;
   sReplace01umFilter.sElement.AlarmThreshold := 4000;
   sReplaceActiveCarbonFilter.sElement.WarningThreshold := 3200;
   sReplaceActiveCarbonFilter.sElement.AlarmThreshold := 4000;
   sUTLExtraction_ReplaceParticleFilter.sElement.WarningThreshold := 3200;
   sUTLExtraction_ReplaceParticleFilter.sElement.AlarmThreshold := 4000;
   sUTLExtraction_ReplaceFilterCassetteAndActiveCarbonFilter.sElement.WarningThreshold := 3200;
   sUTLExtraction_ReplaceFilterCassetteAndActiveCarbonFilter.sElement.AlarmThreshold := 4000;
   sReplaceSealOnSas.sElement.WarningThreshold := 4800;
   sReplaceSealOnSas.sElement.AlarmThreshold := 6000;
   sGreaseAxes.sElement.WarningThreshold := 4800;
   sGreaseAxes.sElement.AlarmThreshold := 6000;
END_DATA_BLOCK

DATA_BLOCK "DB_Temperature"   // DB490
// stored: AutoNumber false, InstanceOfName FB_Temperature, InstanceOfType FB
"FB_Temperature"
BEGIN
END_DATA_BLOCK

DATA_BLOCK "DB_LightsManagement"   // DB500
// stored: AutoNumber false, InstanceOfName FB_LightsManagement, InstanceOfType FB
"FB_LightsManagement"
BEGIN
END_DATA_BLOCK

DATA_BLOCK "DB_MainDoorManagement"   // DB96
// stored: InstanceOfName FB_MainDoorManagement, InstanceOfType FB
"FB_MainDoorManagement"
BEGIN
END_DATA_BLOCK

DATA_BLOCK "DB_WarmUP"   // DB530
// stored: AutoNumber false, InstanceOfName FB_WarmUP, InstanceOfType FB
"FB_WarmUP"
BEGIN
END_DATA_BLOCK

DATA_BLOCK "LBP_AlarmMsgs"   // DB2
TITLE = PLC-Error / Messages / Erreur AP / messages
{ S7_Optimized_Access := 'FALSE' }
AUTHOR : SINUMERIK
FAMILY : SINUMERIK_ONE
VERSION : 6.24
// Interface between user program and LBP_GenAlarmMsgs [FC10], contains bit arrays for blocking and stop signals as well as fault and status messages. / Interface entre programme utilisateur et LBP_GenAlarmMsgs [FC10] contient des tableaux de bits pour bloquer et arrêter des signaux et des signalisations de défaut et d'état.
// stored: AutoNumber false, InstanceOfName LBP_typeAlarmMsgs, InstanceOfType UDT
"LBP_typeAlarmMsgs"
BEGIN
END_DATA_BLOCK

DATA_BLOCK "LBP_Axis01_X"   // DB31
TITLE = Axis-specific signals
{ S7_Optimized_Access := 'FALSE' }
AUTHOR : SINUMERIK
FAMILY : SINUMERIK_ONE
VERSION : 6.14
// Interface between user program and axis/spindle, contains signals from/to axis/spindle 1
// stored: AutoNumber false, InstanceOfName LBP_typeAxisX, InstanceOfType UDT
"LBP_typeAxisX"
BEGIN
END_DATA_BLOCK

DATA_BLOCK "LBP_Axis02_Y"   // DB32
TITLE = Axis-specific signals
{ S7_Optimized_Access := 'FALSE' }
AUTHOR : SINUMERIK
FAMILY : SINUMERIK_ONE
VERSION : 6.14
// Interface between user program and axis/spindle, contains signals from/to axis/spindle 2
// stored: AutoNumber false, InstanceOfName LBP_typeAxisX, InstanceOfType UDT
"LBP_typeAxisX"
BEGIN
END_DATA_BLOCK

DATA_BLOCK "LBP_Axis03_ZM"   // DB33
TITLE = Axis-specific signals
{ S7_Optimized_Access := 'FALSE' }
AUTHOR : SINUMERIK
FAMILY : SINUMERIK_ONE
VERSION : 6.14
// Interface between user program and axis/spindle, contains signals from/to axis/spindle 3
// stored: AutoNumber false, InstanceOfName LBP_typeAxisX, InstanceOfType UDT
"LBP_typeAxisX"
BEGIN
END_DATA_BLOCK

DATA_BLOCK "LBP_Axis04_B"   // DB34
TITLE = Axis-specific signals
{ S7_Optimized_Access := 'FALSE' }
AUTHOR : SINUMERIK
FAMILY : SINUMERIK_ONE
VERSION : 6.14
// Interface between user program and axis/spindle, contains signals from/to axis/spindle 4
// stored: AutoNumber false, InstanceOfName LBP_typeAxisX, InstanceOfType UDT
"LBP_typeAxisX"
BEGIN
END_DATA_BLOCK

DATA_BLOCK "LBP_Axis05_U1"   // DB35
TITLE = Axis-specific signals
{ S7_Optimized_Access := 'FALSE' }
AUTHOR : SINUMERIK
FAMILY : SINUMERIK_ONE
VERSION : 6.14
// Interface between user program and axis/spindle, contains signals from/to axis/spindle 5
// stored: AutoNumber false, InstanceOfName LBP_typeAxisX, InstanceOfType UDT
"LBP_typeAxisX"
BEGIN
END_DATA_BLOCK

DATA_BLOCK "LBP_Axis06_U2"   // DB36
TITLE = Axis-specific signals
{ S7_Optimized_Access := 'FALSE' }
AUTHOR : SINUMERIK
FAMILY : SINUMERIK_ONE
VERSION : 6.14
// Interface between user program and axis/spindle, contains signals from/to axis/spindle 6
// stored: AutoNumber false, InstanceOfName LBP_typeAxisX, InstanceOfType UDT
"LBP_typeAxisX"
BEGIN
END_DATA_BLOCK

DATA_BLOCK "LBP_Axis07_V"   // DB37
TITLE = Axis-specific signals
{ S7_Optimized_Access := 'FALSE' }
AUTHOR : SINUMERIK
FAMILY : SINUMERIK_ONE
VERSION : 6.14
// Interface between user program and axis/spindle, contains signals from/to axis/spindle 7
// stored: AutoNumber false, InstanceOfName LBP_typeAxisX, InstanceOfType UDT
"LBP_typeAxisX"
BEGIN
END_DATA_BLOCK

DATA_BLOCK "LBP_Axis08_W"   // DB38
TITLE = Axis-specific signals
{ S7_Optimized_Access := 'FALSE' }
AUTHOR : SINUMERIK
FAMILY : SINUMERIK_ONE
VERSION : 6.14
// Interface between user program and axis/spindle, contains signals from/to axis/spindle 8
// stored: AutoNumber false, InstanceOfName LBP_typeAxisX, InstanceOfType UDT
"LBP_typeAxisX"
BEGIN
END_DATA_BLOCK

DATA_BLOCK "LBP_Axis09_ZL"   // DB39
TITLE = Axis-specific signals
{ S7_Optimized_Access := 'FALSE' }
AUTHOR : SINUMERIK
FAMILY : SINUMERIK_ONE
VERSION : 6.14
// Interface between user program and axis/spindle, contains signals from/to axis/spindle 9
// stored: AutoNumber false, InstanceOfName LBP_typeAxisX, InstanceOfType UDT
"LBP_typeAxisX"
BEGIN
END_DATA_BLOCK

DATA_BLOCK "LBP_Axis10"   // DB40
TITLE = Axis-specific signals
{ S7_Optimized_Access := 'FALSE' }
AUTHOR : SINUMERIK
FAMILY : SINUMERIK_ONE
VERSION : 6.14
// Interface between user program and axis/spindle, contains signals from/to axis/spindle 10
// stored: AutoNumber false, InstanceOfName LBP_typeAxisX, InstanceOfType UDT
"LBP_typeAxisX"
BEGIN
END_DATA_BLOCK

DATA_BLOCK "LBP_Axis11"   // DB41
TITLE = Axis-specific signals / Signaux spécifiques à un axe
{ S7_Optimized_Access := 'FALSE' }
AUTHOR : SINUMERIK
FAMILY : SINUMERIK_ONE
VERSION : 6.24
// Interface between user program and axis/spindle, contains signals from/to axis/spindle 11 / Interface entre programme utilisateur et axe/broche, contient des signaux de/vers axe/broche 11
// stored: AutoNumber false, InstanceOfName LBP_typeAxisX, InstanceOfType UDT
"LBP_typeAxisX"
BEGIN
END_DATA_BLOCK

DATA_BLOCK "LBP_Axis12"   // DB42
TITLE = Axis-specific signals / Signaux spécifiques à un axe
{ S7_Optimized_Access := 'FALSE' }
AUTHOR : SINUMERIK
FAMILY : SINUMERIK_ONE
VERSION : 6.24
// Interface between user program and axis/spindle, contains signals from/to axis/spindle 12 / Interface entre programme utilisateur et axe/broche, contient des signaux de/vers axe/broche 12
// stored: AutoNumber false, InstanceOfName LBP_typeAxisX, InstanceOfType UDT
"LBP_typeAxisX"
BEGIN
END_DATA_BLOCK

DATA_BLOCK "LBP_Axis13"   // DB43
TITLE = Axis-specific signals / Signaux spécifiques à un axe
{ S7_Optimized_Access := 'FALSE' }
AUTHOR : SINUMERIK
FAMILY : SINUMERIK_ONE
VERSION : 6.24
// Interface between user program and axis/spindle, contains signals from/to axis/spindle 13 / Interface entre programme utilisateur et axe/broche, contient des signaux de/vers axe/broche 13
// stored: AutoNumber false, InstanceOfName LBP_typeAxisX, InstanceOfType UDT
"LBP_typeAxisX"
BEGIN
END_DATA_BLOCK

DATA_BLOCK "LBP_Axis14"   // DB44
TITLE = Axis-specific signals / Signaux spécifiques à un axe
{ S7_Optimized_Access := 'FALSE' }
AUTHOR : SINUMERIK
FAMILY : SINUMERIK_ONE
VERSION : 6.24
// Interface between user program and axis/spindle, contains signals from/to axis/spindle 14 / Interface entre programme utilisateur et axe/broche, contient des signaux de/vers axe/broche 14
// stored: AutoNumber false, InstanceOfName LBP_typeAxisX, InstanceOfType UDT
"LBP_typeAxisX"
BEGIN
END_DATA_BLOCK

DATA_BLOCK "LBP_Axis15"   // DB45
TITLE = Axis-specific signals / Signaux spécifiques à un axe
{ S7_Optimized_Access := 'FALSE' }
AUTHOR : SINUMERIK
FAMILY : SINUMERIK_ONE
VERSION : 6.24
// Interface between user program and axis/spindle, contains signals from/to axis/spindle 15 / Interface entre programme utilisateur et axe/broche, contient des signaux de/vers axe/broche 15
// stored: AutoNumber false, InstanceOfName LBP_typeAxisX, InstanceOfType UDT
"LBP_typeAxisX"
BEGIN
END_DATA_BLOCK

DATA_BLOCK "LBP_Axis16"   // DB46
TITLE = Axis-specific signals / Signaux spécifiques à un axe
{ S7_Optimized_Access := 'FALSE' }
AUTHOR : SINUMERIK
FAMILY : SINUMERIK_ONE
VERSION : 6.24
// Interface between user program and axis/spindle, contains signals from/to axis/spindle 16 / Interface entre programme utilisateur et axe/broche, contient des signaux de/vers axe/broche 16
// stored: AutoNumber false, InstanceOfName LBP_typeAxisX, InstanceOfType UDT
"LBP_typeAxisX"
BEGIN
END_DATA_BLOCK

DATA_BLOCK "LBP_Axis17"   // DB47
TITLE = Axis-specific signals / Signaux spécifiques à un axe
{ S7_Optimized_Access := 'FALSE' }
AUTHOR : SINUMERIK
FAMILY : SINUMERIK_ONE
VERSION : 6.24
// Interface between user program and axis/spindle, contains signals from/to axis/spindle 17 / Interface entre programme utilisateur et axe/broche, contient des signaux de/vers axe/broche 17
// stored: AutoNumber false, InstanceOfName LBP_typeAxisX, InstanceOfType UDT
"LBP_typeAxisX"
BEGIN
END_DATA_BLOCK

DATA_BLOCK "LBP_Axis18"   // DB48
TITLE = Axis-specific signals / Signaux spécifiques à un axe
{ S7_Optimized_Access := 'FALSE' }
AUTHOR : SINUMERIK
FAMILY : SINUMERIK_ONE
VERSION : 6.24
// Interface between user program and axis/spindle, contains signals from/to axis/spindle 18 / Interface entre programme utilisateur et axe/broche, contient des signaux de/vers axe/broche 18
// stored: AutoNumber false, InstanceOfName LBP_typeAxisX, InstanceOfType UDT
"LBP_typeAxisX"
BEGIN
END_DATA_BLOCK

DATA_BLOCK "LBP_Axis19"   // DB49
TITLE = Axis-specific signals / Signaux spécifiques à un axe
{ S7_Optimized_Access := 'FALSE' }
AUTHOR : SINUMERIK
FAMILY : SINUMERIK_ONE
VERSION : 6.24
// Interface between user program and axis/spindle, contains signals from/to axis/spindle 19 / Interface entre programme utilisateur et axe/broche, contient des signaux de/vers axe/broche 19
// stored: AutoNumber false, InstanceOfName LBP_typeAxisX, InstanceOfType UDT
"LBP_typeAxisX"
BEGIN
END_DATA_BLOCK

DATA_BLOCK "LBP_Axis20"   // DB50
TITLE = Axis-specific signals / Signaux spécifiques à un axe
{ S7_Optimized_Access := 'FALSE' }
AUTHOR : SINUMERIK
FAMILY : SINUMERIK_ONE
VERSION : 6.24
// Interface between user program and axis/spindle, contains signals from/to axis/spindle 20 / Interface entre programme utilisateur et axe/broche, contient des signaux de/vers axe/broche 20
// stored: AutoNumber false, InstanceOfName LBP_typeAxisX, InstanceOfType UDT
"LBP_typeAxisX"
BEGIN
END_DATA_BLOCK

DATA_BLOCK "LBP_Axis21"   // DB51
TITLE = Axis-specific signals / Signaux spécifiques à un axe
{ S7_Optimized_Access := 'FALSE' }
AUTHOR : SINUMERIK
FAMILY : SINUMERIK_ONE
VERSION : 6.24
// Interface between user program and axis/spindle, contains signals from/to axis/spindle 21 / Interface entre programme utilisateur et axe/broche, contient des signaux de/vers axe/broche 21
// stored: AutoNumber false, InstanceOfName LBP_typeAxisX, InstanceOfType UDT
"LBP_typeAxisX"
BEGIN
END_DATA_BLOCK

DATA_BLOCK "LBP_Axis22"   // DB52
TITLE = Axis-specific signals / Signaux spécifiques à un axe
{ S7_Optimized_Access := 'FALSE' }
AUTHOR : SINUMERIK
FAMILY : SINUMERIK_ONE
VERSION : 6.24
// Interface between user program and axis/spindle, contains signals from/to axis/spindle 22 / Interface entre programme utilisateur et axe/broche, contient des signaux de/vers axe/broche 22
// stored: AutoNumber false, InstanceOfName LBP_typeAxisX, InstanceOfType UDT
"LBP_typeAxisX"
BEGIN
END_DATA_BLOCK

DATA_BLOCK "LBP_Axis23"   // DB53
TITLE = Axis-specific signals / Signaux spécifiques à un axe
{ S7_Optimized_Access := 'FALSE' }
AUTHOR : SINUMERIK
FAMILY : SINUMERIK_ONE
VERSION : 6.24
// Interface between user program and axis/spindle, contains signals from/to axis/spindle 23 / Interface entre programme utilisateur et axe/broche, contient des signaux de/vers axe/broche 23
// stored: AutoNumber false, InstanceOfName LBP_typeAxisX, InstanceOfType UDT
"LBP_typeAxisX"
BEGIN
END_DATA_BLOCK

DATA_BLOCK "LBP_Axis24"   // DB54
TITLE = Axis-specific signals / Signaux spécifiques à un axe
{ S7_Optimized_Access := 'FALSE' }
AUTHOR : SINUMERIK
FAMILY : SINUMERIK_ONE
VERSION : 6.24
// Interface between user program and axis/spindle, contains signals from/to axis/spindle 24 / Interface entre programme utilisateur et axe/broche, contient des signaux de/vers axe/broche 24
// stored: AutoNumber false, InstanceOfName LBP_typeAxisX, InstanceOfType UDT
"LBP_typeAxisX"
BEGIN
END_DATA_BLOCK

DATA_BLOCK "LBP_Axis25"   // DB55
TITLE = Axis-specific signals / Signaux spécifiques à un axe
{ S7_Optimized_Access := 'FALSE' }
AUTHOR : SINUMERIK
FAMILY : SINUMERIK_ONE
VERSION : 6.24
// Interface between user program and axis/spindle, contains signals from/to axis/spindle 25 / Interface entre programme utilisateur et axe/broche, contient des signaux de/vers axe/broche 25
// stored: AutoNumber false, InstanceOfName LBP_typeAxisX, InstanceOfType UDT
"LBP_typeAxisX"
BEGIN
END_DATA_BLOCK

DATA_BLOCK "LBP_Axis26"   // DB56
TITLE = Axis-specific signals / Signaux spécifiques à un axe
{ S7_Optimized_Access := 'FALSE' }
AUTHOR : SINUMERIK
FAMILY : SINUMERIK_ONE
VERSION : 6.24
// Interface between user program and axis/spindle, contains signals from/to axis/spindle 26 / Interface entre programme utilisateur et axe/broche, contient des signaux de/vers axe/broche 26
// stored: AutoNumber false, InstanceOfName LBP_typeAxisX, InstanceOfType UDT
"LBP_typeAxisX"
BEGIN
END_DATA_BLOCK

DATA_BLOCK "LBP_Axis27"   // DB57
TITLE = Axis-specific signals / Signaux spécifiques à un axe
{ S7_Optimized_Access := 'FALSE' }
AUTHOR : SINUMERIK
FAMILY : SINUMERIK_ONE
VERSION : 6.24
// Interface between user program and axis/spindle, contains signals from/to axis/spindle 27 / Interface entre programme utilisateur et axe/broche, contient des signaux de/vers axe/broche 27
// stored: AutoNumber false, InstanceOfName LBP_typeAxisX, InstanceOfType UDT
"LBP_typeAxisX"
BEGIN
END_DATA_BLOCK

DATA_BLOCK "LBP_Axis28"   // DB58
TITLE = Axis-specific signals / Signaux spécifiques à un axe
{ S7_Optimized_Access := 'FALSE' }
AUTHOR : SINUMERIK
FAMILY : SINUMERIK_ONE
VERSION : 6.24
// Interface between user program and axis/spindle, contains signals from/to axis/spindle 28 / Interface entre programme utilisateur et axe/broche, contient des signaux de/vers axe/broche 28
// stored: AutoNumber false, InstanceOfName LBP_typeAxisX, InstanceOfType UDT
"LBP_typeAxisX"
BEGIN
END_DATA_BLOCK

DATA_BLOCK "LBP_Axis29"   // DB59
TITLE = Axis-specific signals / Signaux spécifiques à un axe
{ S7_Optimized_Access := 'FALSE' }
AUTHOR : SINUMERIK
FAMILY : SINUMERIK_ONE
VERSION : 6.24
// Interface between user program and axis/spindle, contains signals from/to axis/spindle 29 / Interface entre programme utilisateur et axe/broche, contient des signaux de/vers axe/broche 29
// stored: AutoNumber false, InstanceOfName LBP_typeAxisX, InstanceOfType UDT
"LBP_typeAxisX"
BEGIN
END_DATA_BLOCK

